# B&R Automation Studio project OpcUaSample410_BrbLibUa103 (part 14)

#### BrbUaRsGetEvent.c
```c
#include <bur/plctypes.h>
#ifdef __cplusplus
	extern "C"
	{
#endif

#include "BrbLibUa.h"
#include <string.h>
#include <AnsiCFunc.h>

#ifdef __cplusplus
	};
#endif

// NOLINTBEGIN(readability-*, bugprone-easily-swappable-parameters, bugprone-branch-clone, clang-diagnostic-invalid-utf8, clang-diagnostic-invalid-source-encoding, clang-diagnostic-pointer-arith, clang-diagnostic-strict-prototypes, hicpp-uppercase-literal-suffix, cppcoreguidelines-*, performance-*)

/* Gibt ein ermitteltes Event zurück */
unsigned short BrbUaRsGetEvent(struct BrbUaRunServer_TYP* pRunServer, unsigned short nEventIndex, struct BrbUaRsEvent_TYP* pEvent, struct BrbUaRsEventIntern_TYP* pEventIntern)
{
	UINT nStatus = eBRB_ERR_NULL_POINTER;
	if(pRunServer != 0 && pEvent != 0)
	{
		memset(pEvent, 0, sizeof(BrbUaRsEvent_TYP));
		nStatus = eBRB_ERR_UA_NO_ELEMENTS;
		if(pRunServer->Events.nEventCount > 0 && pRunServer->Events.pEvents != 0)
		{
			nStatus = eBRB_ERR_UA_INVALID_INDEX;
			if(nEventIndex < pRunServer->Events.nEventCount)
			{
				nStatus = eBRB_ERR_OK;
				BrbUaRsEventIntern_TYP* pEventInternOri = ((BrbUaRsEventIntern_TYP*)pRunServer->Events.pEvents) + nEventIndex;
				pEvent->nFieldCount = pEventInternOri->nFieldCount;
				memcpy(&pEvent->TypeNodeId, &pEventInternOri->TypeNodeId, sizeof(UANodeID));
				if(pEventIntern != 0)
				{
					memcpy(pEventIntern, pEventInternOri, sizeof(BrbUaRsEventIntern_TYP));
				}
			}
		}
	}
	return nStatus;
}

// NOLINTEND(readability-*, bugprone-easily-swappable-parameters, bugprone-branch-clone, clang-diagnostic-invalid-utf8, clang-diagnostic-invalid-source-encoding, clang-diagnostic-pointer-arith, clang-diagnostic-strict-prototypes, hicpp-uppercase-literal-suffix, cppcoreguidelines-*, performance-*)
```

#### BrbUaRsGetEventField.c
```c
#include <bur/plctypes.h>
#ifdef __cplusplus
	extern "C"
	{
#endif

#include "BrbLibUa.h"
#include <string.h>
#include <AnsiCFunc.h>

#ifdef __cplusplus
	};
#endif

// NOLINTBEGIN(readability-*, bugprone-easily-swappable-parameters, bugprone-branch-clone, clang-diagnostic-invalid-utf8, clang-diagnostic-invalid-source-encoding, clang-diagnostic-pointer-arith, clang-diagnostic-strict-prototypes, hicpp-uppercase-literal-suffix, cppcoreguidelines-*, performance-*)

/* Gibt ein ermitteltes Field zurück */
unsigned short BrbUaRsGetEventField(struct BrbUaRunServer_TYP* pRunServer, unsigned short nEventIndex, unsigned short nEventFieldIndex, struct UaSrv_FireEventFieldType* pEventField)
{
	UINT nStatus = eBRB_ERR_NULL_POINTER;
	if(pRunServer != 0 && pEventField != 0)
	{
		memset(pEventField, 0, sizeof(UaSrv_FireEventFieldType));
		nStatus = eBRB_ERR_UA_NO_ELEMENTS;
		if(pRunServer->Events.nEventCount > 0 && pRunServer->Events.pEvents != 0)
		{
			nStatus = eBRB_ERR_UA_INVALID_INDEX;
			if(nEventIndex < pRunServer->Events.nEventCount)
			{
				nStatus = eBRB_ERR_UA_NO_ELEMENTS;
				BrbUaRsEventIntern_TYP* pEventIntern = ((BrbUaRsEventIntern_TYP*)pRunServer->Events.pEvents) + nEventIndex;
				if(pEventIntern->nFieldCount > 0 && pEventIntern->pFields)
				{
					nStatus = eBRB_ERR_UA_INVALID_INDEX;
					if(nEventFieldIndex < pEventIntern->nFieldCount)
					{
						nStatus = eBRB_ERR_OK;
						UaSrv_FireEventFieldType* pEventFieldOri = ((UaSrv_FireEventFieldType*)pEventIntern->pFields) + nEventFieldIndex;
						memcpy(pEventField, pEventFieldOri, sizeof(UaSrv_FireEventFieldType));
					}
				}
			}
		}
	}
	return nStatus;
}

// NOLINTEND(readability-*, bugprone-easily-swappable-parameters, bugprone-branch-clone, clang-diagnostic-invalid-utf8, clang-diagnostic-invalid-source-encoding, clang-diagnostic-pointer-arith, clang-diagnostic-strict-prototypes, hicpp-uppercase-literal-suffix, cppcoreguidelines-*, performance-*)
```

#### BrbUaRsMonitor.c
```c
#include <bur/plctypes.h>
#ifdef __cplusplus
	extern "C"
	{
#endif

#include "BrbLibUa.h"
#include <string.h>
#include <AnsiCFunc.h>

#ifdef __cplusplus
	};
#endif

// NOLINTBEGIN(readability-*, bugprone-easily-swappable-parameters, bugprone-branch-clone, clang-diagnostic-invalid-utf8, clang-diagnostic-invalid-source-encoding, clang-diagnostic-pointer-arith, clang-diagnostic-strict-prototypes, hicpp-uppercase-literal-suffix, cppcoreguidelines-*, performance-*)

/* Zeigt die Inhalte des internen Speichers */
unsigned short BrbUaRsMonitor(struct BrbUaRunServer_TYP* pRunServer, struct BrbUaRsMonitor_TYP* pMonitor)
{
	UINT nStatus = eBRB_ERR_NULL_POINTER;
	if(pRunServer != 0 && pMonitor != 0)
	{
		nStatus = eBRB_ERR_NOT_ENABLED;
		if(pMonitor->bEnable == 1)
		{
			nStatus = eBRB_ERR_OK;
			brsmemset((UDINT)&pMonitor->Namespace.Namespace, 0, sizeof(pMonitor->Namespace.Namespace));
			BrbUaRsGetNamespace(pRunServer, pMonitor->Namespace.nDatObjNamespaceIndex, &pMonitor->Namespace.Namespace);

			brsmemset((UDINT)&pMonitor->Event.Event, 0, sizeof(pMonitor->Event.Event));
			brsmemset((UDINT)&pMonitor->Event.EventIntern, 0, sizeof(pMonitor->Event.EventIntern));
			pMonitor->Event.nMonitorStatus = BrbUaRsGetEvent(pRunServer, pMonitor->Event.nEventIndex, &pMonitor->Event.Event, &pMonitor->Event.EventIntern);

			brsmemset((UDINT)&pMonitor->EventField.Field, 0, sizeof(pMonitor->EventField.Field));
			pMonitor->EventField.nMonitorStatus = BrbUaRsGetEventField(pRunServer, pMonitor->EventField.nEventIndex, pMonitor->EventField.nEventFieldIndex, &pMonitor->EventField.Field);
		}
		else
		{
			brsmemset((UDINT)&pMonitor->Namespace.Namespace, 0, sizeof(pMonitor->Namespace.Namespace));
			pMonitor->Event.nMonitorStatus = eBRB_ERR_NOT_ENABLED;
			brsmemset((UDINT)&pMonitor->Event.Event, 0, sizeof(pMonitor->Event.Event));
			brsmemset((UDINT)&pMonitor->Event.EventIntern, 0, sizeof(pMonitor->Event.EventIntern));
			pMonitor->EventField.nMonitorStatus = eBRB_ERR_NOT_ENABLED;
			brsmemset((UDINT)&pMonitor->EventField.Field, 0, sizeof(pMonitor->EventField.Field));
		}
		pMonitor->nMonitorStatus = nStatus;
	}
	return nStatus;
}

// NOLINTEND(readability-*, bugprone-easily-swappable-parameters, bugprone-branch-clone, clang-diagnostic-invalid-utf8, clang-diagnostic-invalid-source-encoding, clang-diagnostic-pointer-arith, clang-diagnostic-strict-prototypes, hicpp-uppercase-literal-suffix, cppcoreguidelines-*, performance-*)
```

- Project.language (not shown)

### ReadMe.txt
```
Die AS-Solution 'UnitTest' ist eine Unterstützung für wiederholbare Aufruf-Tests.
Dabei sind Test-Routinen implementiert, welche ihrerseits Bibliotheks-Funktionen mit definierten Eingangs-Werten aufrufen,
die zurückgegebenen Ausgänge prüfen und so einen Bericht erstellen. Entspricht ein Ausgang nicht dem erwarteten Ergebnis,
wird dies im Bericht vermerkt.
Das Aufrufen aller Test-Routinen kann mit wenigen Mausklicks ausgeführt werden. So kann nach Änderung oder Erweiterung einer
Funktion sehr schnell deren Kompatibilität und Funktionstüchtigkeit geprüft werden, was zu einer Erhöhung der SW-Qualität führt.
Für das Beispiel zur Nutzung der geprüften Bibliothek sind die UnitTests nicht von Belang.
```

### Package Logical/UnitTests/UnitTestLibraries - Libraries for asserts

### Library Logical/UnitTests/UnitTestLibraries/BrbAsserts (ANSIC) - Brb custom asserts

#### BrbAsserts.h - Include this file in programs using any of the asserts provided by this library
```c
/********************************************************************
 * COPYRIGHT -- Bernecker + Rainer
 ********************************************************************
 * Library: BrbAsserts
 * File: BrbAsserts.h
 * Author: Rainer Niedermeier
 *******************************************************************/

#include <bur/plctypes.h>
#include "UnitTest.h"

/* When this file is included the defines, makros  of the following header files should be provided as well:  */
#include "EqualBool.h"
#include "EqualDint.h"
#include "EqualUdint.h"
#include "EqualDtStruct.h"
#include "WithinUdint.h"
#include "WithinDint.h"
#include "MemContent.h"
#include "StringEndContent.h"
```

#### EqualBool.h
```c
/********************************************************************
 * COPYRIGHT -- Bernecker + Rainer
 ********************************************************************
 * Library: BrbAsserts
 * File: EqualBool.c
 * Author: Rainer Niedermeier
 *******************************************************************/

#include <bur/plctypes.h>
#include "UnitTest.h"

#ifdef __cplusplus
extern "C"
{
#endif

// NOLINTBEGIN(readability-*, bugprone-easily-swappable-parameters, clang-diagnostic-invalid-utf8, clang-diagnostic-invalid-source-encoding, clang-diagnostic-pointer-arith, clang-diagnostic-strict-prototypes, hicpp-uppercase-literal-suffix, cppcoreguidelines-*, performance-*, readability-avoid-const-params-in-decls)

/* Dummies for smart edit autocompletion.
See below for the real macros used by the compiler  */
#ifdef _SMART_EDIT_DUMMY_
	/* Returns true if they are equal. */
	BOOL BRB_ASSERT_EQUAL_BOOL(const BOOL expected, const BOOL actual);
#endif

/* Prototyping of functions.
These declaration of functions are used by the compiler to check number and type of arguments. */
BOOL brb_assertEqualBool(const BOOL expected, const BOOL actual, unsigned long line, const char *file);

/* Macros used in the test implementation.
The macro passes the location information to the implemented assert. */
#define BRB_ASSERT_EQUAL_BOOL(expected, actual) brb_assertEqualBool(expected, actual, (unsigned long) __LINE__, __FILE__)

// NOLINTEND(readability-*, bugprone-easily-swappable-parameters, clang-diagnostic-invalid-utf8, clang-diagnostic-invalid-source-encoding, clang-diagnostic-pointer-arith, clang-diagnostic-strict-prototypes, hicpp-uppercase-literal-suffix, cppcoreguidelines-*, performance-*, readability-avoid-const-params-in-decls)

#ifdef __cplusplus
};
#endif
```

#### EqualBool.c
```c
/********************************************************************
 * COPYRIGHT -- Bernecker + Rainer
 ********************************************************************
 * Library: BrbAsserts
 * File: EqualBool.c
 * Author: Rainer Niedermeier
 *******************************************************************/

#include <bur/plctypes.h>
#include "BrbAsserts.h"
#include "AsBrStr.h"
#include "BrbLib.h"

#define TRUE 1
#define FALSE 0

// NOLINTBEGIN(readability-*, bugprone-easily-swappable-parameters, bugprone-branch-clone, clang-diagnostic-invalid-utf8, clang-diagnostic-invalid-source-encoding, clang-diagnostic-pointer-arith, clang-diagnostic-strict-prototypes, clang-diagnostic-bad-function-cast, clang-analyzer-security.insecureAPI.*, hicpp-uppercase-literal-suffix, cppcoreguidelines-*, performance-*)
BOOL brb_assertEqualBool(const BOOL expected, const BOOL actual,
	unsigned long line, const char *file)
{
	STRING buffer[100];
	STRING numbuf[15];
	BOOL result = TRUE;
	if(expected == actual)
	{
		addPassed("", line, file);
	}
	else
	{
		brsstrcpy((unsigned long) buffer, (unsigned long) "expected bool ");
		brsitoa((DINT)expected, (UDINT)&numbuf);
		brsstrcat((unsigned long) buffer, (unsigned long) numbuf);
		brsstrcat((unsigned long) buffer, (unsigned long) " was ");
		brsitoa((DINT)actual, (UDINT)&numbuf);
		brsstrcat((unsigned long) buffer, (unsigned long) numbuf);
		addFailure(buffer, line, file);
		result = FALSE;
	}
	return result;
}

// NOLINTEND(readability-*, bugprone-easily-swappable-parameters, bugprone-branch-clone, clang-diagnostic-invalid-utf8, clang-diagnostic-invalid-source-encoding, clang-diagnostic-pointer-arith, clang-diagnostic-strict-prototypes, clang-diagnostic-bad-function-cast, clang-analyzer-security.insecureAPI.*, hicpp-uppercase-literal-suffix, cppcoreguidelines-*, performance-*)
```

#### EqualDint.h
```c
/********************************************************************
 * COPYRIGHT -- Bernecker + Rainer
 ********************************************************************
 * Library: BrbAsserts
 * File: EqualDint.c
 * Author: Rainer Niedermeier
 *******************************************************************/

#include <bur/plctypes.h>
#include "UnitTest.h"

#ifdef __cplusplus
extern "C"
{
#endif

// NOLINTBEGIN(readability-*, bugprone-easily-swappable-parameters, clang-diagnostic-invalid-utf8, clang-diagnostic-invalid-source-encoding, clang-diagnostic-pointer-arith, clang-diagnostic-strict-prototypes, hicpp-uppercase-literal-suffix, cppcoreguidelines-*, performance-*, readability-avoid-const-params-in-decls)

/* Dummies for smart edit autocompletion.
See below for the real macros used by the compiler  */
#ifdef _SMART_EDIT_DUMMY_
	/* Returns true if they are equal. */
	BOOL BRB_ASSERT_EQUAL_DINT(const DINT expected, const DINT actual);
#endif

/* Prototyping of functions.
These declaration of functions are used by the compiler to check number and type of arguments. */
BOOL brb_assertEqualDint(const DINT expected, const DINT actual, unsigned long line, const char *file);

/* Macros used in the test implementation.
The macro passes the location information to the implemented assert. */
#define BRB_ASSERT_EQUAL_DINT(expected, actual) brb_assertEqualDint(expected, actual, (unsigned long) __LINE__, __FILE__)

// NOLINTEND(readability-*, bugprone-easily-swappable-parameters, clang-diagnostic-invalid-utf8, clang-diagnostic-invalid-source-encoding, clang-diagnostic-pointer-arith, clang-diagnostic-strict-prototypes, hicpp-uppercase-literal-suffix, cppcoreguidelines-*, performance-*, readability-avoid-const-params-in-decls)

#ifdef __cplusplus
};
#endif
```

#### EqualDint.c
```c
/********************************************************************
 * COPYRIGHT -- Bernecker + Rainer
 ********************************************************************
 * Library: BrbAsserts
 * File: EqualDint.c
 * Author: Rainer Niedermeier
 *******************************************************************/

#include <bur/plctypes.h>
#include "BrbAsserts.h"
#include "AsBrStr.h"
#include "BrbLib.h"

#define TRUE 1
#define FALSE 0

// NOLINTBEGIN(readability-*, bugprone-easily-swappable-parameters, bugprone-branch-clone, clang-diagnostic-invalid-utf8, clang-diagnostic-invalid-source-encoding, clang-diagnostic-pointer-arith, clang-diagnostic-strict-prototypes, clang-diagnostic-bad-function-cast, clang-analyzer-security.insecureAPI.*, hicpp-uppercase-literal-suffix, cppcoreguidelines-*, performance-*)
BOOL brb_assertEqualDint(const DINT expected, const DINT actual,
	unsigned long line, const char *file)
{
	STRING buffer[100];
	STRING numbuf[15];
	BOOL result = TRUE;
	if(expected == actual)
	{
		addPassed("", line, file);
	}
	else
	{
		brsstrcpy((unsigned long) buffer, (unsigned long) "expected dint ");
		brsitoa((DINT)expected, (UDINT)&numbuf);
		brsstrcat((unsigned long) buffer, (unsigned long) numbuf);
		brsstrcat((unsigned long) buffer, (unsigned long) " was ");
		brsitoa((DINT)actual, (UDINT)&numbuf);
		brsstrcat((unsigned long) buffer, (unsigned long) numbuf);
		addFailure(buffer, line, file);
		result = FALSE;
	}
	return result;
}

// NOLINTEND(readability-*, bugprone-easily-swappable-parameters, bugprone-branch-clone, clang-diagnostic-invalid-utf8, clang-diagnostic-invalid-source-encoding, clang-diagnostic-pointer-arith, clang-diagnostic-strict-prototypes, clang-diagnostic-bad-function-cast, clang-analyzer-security.insecureAPI.*, hicpp-uppercase-literal-suffix, cppcoreguidelines-*, performance-*)
```

#### EqualUdint.h
```c
/********************************************************************
 * COPYRIGHT -- Bernecker + Rainer
 ********************************************************************
 * Library: BrbAsserts
 * File: EqualUdint.c
 * Author: Rainer Niedermeier
 *******************************************************************/

#include <bur/plctypes.h>
#include "UnitTest.h"

#ifdef __cplusplus
extern "C"
{
#endif

// NOLINTBEGIN(readability-*, bugprone-easily-swappable-parameters, clang-diagnostic-invalid-utf8, clang-diagnostic-invalid-source-encoding, clang-diagnostic-pointer-arith, clang-diagnostic-strict-prototypes, hicpp-uppercase-literal-suffix, cppcoreguidelines-*, performance-*, readability-avoid-const-params-in-decls)

/* Dummies for smart edit autocompletion.
See below for the real macros used by the compiler  */
#ifdef _SMART_EDIT_DUMMY_
	/* Returns true if they are equal. */
	BOOL BRB_ASSERT_EQUAL_UDINT(const UDINT expected, const UDINT actual);
#endif

/* Prototyping of functions.
These declaration of functions are used by the compiler to check number and type of arguments. */
BOOL brb_assertEqualUdint(const UDINT expected, const UDINT actual, unsigned long line, const char *file);

/* Macros used in the test implementation.
The macro passes the location information to the implemented assert. */
#define BRB_ASSERT_EQUAL_UDINT(expected, actual) brb_assertEqualUdint(expected, actual, (unsigned long) __LINE__, __FILE__)

// NOLINTEND(readability-*, bugprone-easily-swappable-parameters, clang-diagnostic-invalid-utf8, clang-diagnostic-invalid-source-encoding, clang-diagnostic-pointer-arith, clang-diagnostic-strict-prototypes, hicpp-uppercase-literal-suffix, cppcoreguidelines-*, performance-*, readability-avoid-const-params-in-decls)

#ifdef __cplusplus
};
#endif
```

#### EqualUdint.c
```c
/********************************************************************
 * COPYRIGHT -- Bernecker + Rainer
 ********************************************************************
 * Library: BrbAsserts
 * File: EqualUdint.c
 * Author: Rainer Niedermeier
 *******************************************************************/

#include <bur/plctypes.h>
#include "BrbAsserts.h"
#include "AsBrStr.h"
#include "BrbLib.h"

#define TRUE 1
#define FALSE 0

// NOLINTBEGIN(readability-*, bugprone-easily-swappable-parameters, bugprone-branch-clone, clang-diagnostic-invalid-utf8, clang-diagnostic-invalid-source-encoding, clang-diagnostic-pointer-arith, clang-diagnostic-strict-prototypes, clang-diagnostic-bad-function-cast, clang-analyzer-security.insecureAPI.*, hicpp-uppercase-literal-suffix, cppcoreguidelines-*, performance-*)
BOOL brb_assertEqualUdint(const UDINT expected, const UDINT actual,
	unsigned long line, const char *file)
{
	STRING buffer[100];
	STRING numbuf[15];

	BOOL result = TRUE;
	if(expected == actual)
	{
		addPassed("", line, file);
	}
	else
	{
		brsstrcpy((unsigned long) buffer, (unsigned long) "expected udint ");
		BrbUdintToAscii(expected, numbuf);
		brsstrcat((unsigned long) buffer, (unsigned long) numbuf);
		brsstrcat((unsigned long) buffer, (unsigned long) " was ");
		BrbUdintToAscii(actual, numbuf);
		brsstrcat((unsigned long) buffer, (unsigned long) numbuf);
		addFailure(buffer, line, file);
		result = FALSE;
	}
	return result;
}

// NOLINTEND(readability-*, bugprone-easily-swappable-parameters, bugprone-branch-clone, clang-diagnostic-invalid-utf8, clang-diagnostic-invalid-source-encoding, clang-diagnostic-pointer-arith, clang-diagnostic-strict-prototypes, clang-diagnostic-bad-function-cast, clang-analyzer-security.insecureAPI.*, hicpp-uppercase-literal-suffix, cppcoreguidelines-*, performance-*)
```

#### EqualDtStruct.h
```c
/********************************************************************
 * COPYRIGHT -- Bernecker + Rainer
 ********************************************************************
 * Library: BrbAsserts
 * File: Equal_Udint.h
 * Author: Rainer Niedermeier
 *******************************************************************/

#include <bur/plctypes.h>
#include "UnitTest.h"
#include "AsTime.h" // NOLINT(clang-diagnostic-nonportable-system-include-path)

#ifdef __cplusplus
extern "C"
{
#endif

// NOLINTBEGIN(readability-*, bugprone-easily-swappable-parameters, clang-diagnostic-invalid-utf8, clang-diagnostic-invalid-source-encoding, clang-diagnostic-pointer-arith, clang-diagnostic-strict-prototypes, hicpp-uppercase-literal-suffix, cppcoreguidelines-*, performance-*, readability-avoid-const-params-in-decls)

/* Dummies for smart edit autocompletion.
See below for the real macros used by the compiler  */
#ifdef _SMART_EDIT_DUMMY_
	/* Returns true if they are equal. */
	BOOL BRB_ASSERT_EQUAL_DTSTRUCT(const UINT expectedYear, const USINT expectedMonth, const USINT expectedDay, const USINT expectedWeekday, const USINT expectedHour, const USINT expectedMinute, const USINT expectedSecond, const USINT expectedMilliSecond, const USINT expectedMicroSecond, const DTStructure* actual);
#endif

/* Prototyping of functions.
These declaration of functions are used by the compiler to check number and type of arguments. */
BOOL brb_assertEqualDtStruct(const UINT expectedYear, const USINT expectedMonth, const USINT expectedDay, const USINT expectedWeekday, const USINT expectedHour, const USINT expectedMinute, const USINT expectedSecond, const UINT expectedMilliSecond, const UINT expectedMicroSecond, const DTStructure* actual, unsigned long line, const char *file);

/* Macros used in the test implementation.
The macro passes the location information to the implemented assert. */
#define BRB_ASSERT_EQUAL_DTSTRUCT(expectedYear, expectedMonth, expectedDay, expectedWeekday, expectedHour, expectedMinute, expectedSecond, expectedMilliSecond, expectedMicroSecond, actual) brb_assertEqualDtStruct(expectedYear, expectedMonth, expectedDay, expectedWeekday, expectedHour, expectedMinute, expectedSecond, expectedMilliSecond, expectedMicroSecond, actual, (unsigned long) __LINE__, __FILE__)

// NOLINTEND(readability-*, bugprone-easily-swappable-parameters, clang-diagnostic-invalid-utf8, clang-diagnostic-invalid-source-encoding, clang-diagnostic-pointer-arith, clang-diagnostic-strict-prototypes, hicpp-uppercase-literal-suffix, cppcoreguidelines-*, performance-*, readability-avoid-const-params-in-decls)

#ifdef __cplusplus
};
#endif
```

#### EqualDtStruct.c
```c
/********************************************************************
 * COPYRIGHT -- Bernecker + Rainer
 ********************************************************************
 * Library: BrbAsserts
 * File: Equal_Udint.c
 * Author: Rainer Niedermeier
 *******************************************************************/

#include <bur/plctypes.h>
#include "AsBrStr.h"
#include "EqualDtStruct.h"

#define TRUE 1
#define FALSE 0

// NOLINTBEGIN(readability-*, bugprone-easily-swappable-parameters, bugprone-branch-clone, clang-diagnostic-invalid-utf8, clang-diagnostic-invalid-source-encoding, clang-diagnostic-pointer-arith, clang-diagnostic-strict-prototypes, clang-diagnostic-bad-function-cast, clang-analyzer-security.insecureAPI.*, hicpp-uppercase-literal-suffix, cppcoreguidelines-*, performance-*)
BOOL brb_assertEqualDtStruct(const UINT expectedYear, const USINT expectedMonth, const USINT expectedDay, const USINT expectedWeekday,
														const USINT expectedHour, const USINT expectedMinute, const USINT expectedSecond,
														const UINT expectedMilliSecond, const UINT expectedMicroSecond,
														const DTStructure* actual,
                         		unsigned long line, const char *file)
{
	STRING buffer[100];
	STRING numbuf[15];
	BOOL result = TRUE;
	// year
	if(expectedYear == actual->year)
	{
		addPassed("", line, file);
	}
	else
	{
		brsstrcpy((unsigned long) buffer, (unsigned long) "expected year ");
		brsitoa((int)expectedYear, (unsigned long)numbuf);
		brsstrcat((unsigned long) buffer, (unsigned long) numbuf);
		brsstrcat((unsigned long) buffer, (unsigned long) " was ");
		brsitoa((int)actual->year, (unsigned long)numbuf);
		brsstrcat((unsigned long) buffer, (unsigned long) numbuf);
		addFailure(buffer, line, file);
		result = FALSE;
	}
	// month
	if(expectedMonth == actual->month)
	{
		addPassed("", line, file);
	}
	else
	{
		brsstrcpy((unsigned long) buffer, (unsigned long) "expected month ");
		brsitoa((int)expectedMonth, (unsigned long)numbuf);
		brsstrcat((unsigned long) buffer, (unsigned long) numbuf);
		brsstrcat((unsigned long) buffer, (unsigned long) " was ");
		brsitoa((int)actual->month, (unsigned long)numbuf);
		brsstrcat((unsigned long) buffer, (unsigned long) numbuf);
		addFailure(buffer, line, file);
		result = FALSE;
	}
	// day
	if(expectedDay == actual->day)
	{
		addPassed("", line, file);
	}
	else
	{
		brsstrcpy((unsigned long) buffer, (unsigned long) "expected day ");
		brsitoa((int)expectedDay, (unsigned long)numbuf);
		brsstrcat((unsigned long) buffer, (unsigned long) numbuf);
		brsstrcat((unsigned long) buffer, (unsigned long) " was ");
		brsitoa((int)actual->day, (unsigned long)numbuf);
		brsstrcat((unsigned long) buffer, (unsigned long) numbuf);
		addFailure(buffer, line, file);
		result = FALSE;
	}
	// weekday
	if(expectedWeekday == actual->wday)
	{
		addPassed("", line, file);
	}
	else
	{
		brsstrcpy((unsigned long) buffer, (unsigned long) "expected weekday ");
		brsitoa((int)expectedWeekday, (unsigned long)numbuf);
		brsstrcat((unsigned long) buffer, (unsigned long) numbuf);
		brsstrcat((unsigned long) buffer, (unsigned long) " was ");
		brsitoa((int)actual->wday, (unsigned long)numbuf);
		brsstrcat((unsigned long) buffer, (unsigned long) numbuf);
		addFailure(buffer, line, file);
		result = FALSE;
	}
	// hour
	if(expectedHour == actual->hour)
	{
		addPassed("", line, file);
	}
	else
	{
		brsstrcpy((unsigned long) buffer, (unsigned long) "expected hour ");
		brsitoa((int)expectedHour, (unsigned long)numbuf);
		brsstrcat((unsigned long) buffer, (unsigned long) numbuf);
		brsstrcat((unsigned long) buffer, (unsigned long) " was ");
		brsitoa((int)actual->hour, (unsigned long)numbuf);
		brsstrcat((unsigned long) buffer, (unsigned long) numbuf);
		addFailure(buffer, line, file);
		result = FALSE;
	}
	// minute
	if(expectedMinute == actual->minute)
	{
		addPassed("", line, file);
	}
	else
	{
		brsstrcpy((unsigned long) buffer, (unsigned long) "expected minute ");
		brsitoa((int)expectedMinute, (unsigned long)numbuf);
		brsstrcat((unsigned long) buffer, (unsigned long) numbuf);
		brsstrcat((unsigned long) buffer, (unsigned long) " was ");
		brsitoa((int)actual->minute, (unsigned long)numbuf);
		brsstrcat((unsigned long) buffer, (unsigned long) numbuf);
		addFailure(buffer, line, file);
		result = FALSE;
	}
	// second
	if(expectedSecond == actual->second)
	{
		addPassed("", line, file);
	}
	else
	{
		brsstrcpy((unsigned long) buffer, (unsigned long) "expected second ");
		brsitoa((int)expectedSecond, (unsigned long)numbuf);
		brsstrcat((unsigned long) buffer, (unsigned long) numbuf);
		brsstrcat((unsigned long) buffer, (unsigned long) " was ");
		brsitoa((int)actual->second, (unsigned long)numbuf);
		brsstrcat((unsigned long) buffer, (unsigned long) numbuf);
		addFailure(buffer, line, file);
		result = FALSE;
	}
	// millisecond
	if(expectedMilliSecond == actual->millisec)
	{
		addPassed("", line, file);
	}
	else
	{
		brsstrcpy((unsigned long) buffer, (unsigned long) "expected millisecond ");
		brsitoa((int)expectedMilliSecond, (unsigned long)numbuf);
		brsstrcat((unsigned long) buffer, (unsigned long) numbuf);
		brsstrcat((unsigned long) buffer, (unsigned long) " was ");
		brsitoa((int)actual->millisec, (unsigned long)numbuf);
		brsstrcat((unsigned long) buffer, (unsigned long) numbuf);
		addFailure(buffer, line, file);
		result = FALSE;
	}
	// microsecond
	if(expectedMicroSecond == actual->microsec)
	{
		addPassed("", line, file);
	}
	else
	{
		brsstrcpy((unsigned long) buffer, (unsigned long) "expected microsecond ");
		brsitoa((int)expectedMicroSecond, (unsigned long)numbuf);
		brsstrcat((unsigned long) buffer, (unsigned long) numbuf);
		brsstrcat((unsigned long) buffer, (unsigned long) " was ");
		brsitoa((int)actual->microsec, (unsigned long)numbuf);
		brsstrcat((unsigned long) buffer, (unsigned long) numbuf);
		addFailure(buffer, line, file);
		result = FALSE;
	}
	return result;
}

// NOLINTEND(readability-*, bugprone-easily-swappable-parameters, bugprone-branch-clone, clang-diagnostic-invalid-utf8, clang-diagnostic-invalid-source-encoding, clang-diagnostic-pointer-arith, clang-diagnostic-strict-prototypes, clang-diagnostic-bad-function-cast, clang-analyzer-security.insecureAPI.*, hicpp-uppercase-literal-suffix, cppcoreguidelines-*, performance-*)
```

#### WithinUdint.h
```c
/********************************************************************
 * COPYRIGHT -- Bernecker + Rainer
 ********************************************************************
 * Library: BrbAsserts
 * File: Equal_Udint.h
 * Author: Rainer Niedermeier
 *******************************************************************/

#include <bur/plctypes.h>
#include "UnitTest.h"

#ifdef __cplusplus
extern "C"
{
#endif

// NOLINTBEGIN(readability-*, bugprone-easily-swappable-parameters, clang-diagnostic-invalid-utf8, clang-diagnostic-invalid-source-encoding, clang-diagnostic-pointer-arith, clang-diagnostic-strict-prototypes, hicpp-uppercase-literal-suffix, cppcoreguidelines-*, performance-*, readability-avoid-const-params-in-decls)

/* Dummies for smart edit autocompletion.
See below for the real macros used by the compiler  */
#ifdef _SMART_EDIT_DUMMY_
	/* Returns true if they are equal. */
	BOOL BRB_ASSERT_WITHIN_UDINT(const UDINT min, const UDINT max, const UDINT actual);
#endif

/* Prototyping of functions.
These declaration of functions are used by the compiler to check number and type of arguments. */
BOOL brb_assertWithinUdint(const UDINT min, const UDINT max, const UDINT actual, unsigned long line, const char *file);

/* Macros used in the test implementation.
The macro passes the location information to the implemented assert. */
#define BRB_ASSERT_WITHIN_UDINT(min, max, actual) brb_assertWithinUdint(min, max, actual, (unsigned long) __LINE__, __FILE__)

// NOLINTEND(readability-*, bugprone-easily-swappable-parameters, clang-diagnostic-invalid-utf8, clang-diagnostic-invalid-source-encoding, clang-diagnostic-pointer-arith, clang-diagnostic-strict-prototypes, hicpp-uppercase-literal-suffix, cppcoreguidelines-*, performance-*, readability-avoid-const-params-in-decls)

#ifdef __cplusplus
};
#endif
```

#### WithinUdint.c
```c
/********************************************************************
 * COPYRIGHT -- Bernecker + Rainer
 ********************************************************************
 * Library: BrbAsserts
 * File: Equal_Udint.c
 * Author: Rainer Niedermeier
 *******************************************************************/

#include <bur/plctypes.h>
#include "AsBrStr.h"
#include "BrbLib.h"
#include "WithinUdint.h"

#define TRUE 1
#define FALSE 0

// NOLINTBEGIN(readability-*, bugprone-easily-swappable-parameters, bugprone-branch-clone, clang-diagnostic-invalid-utf8, clang-diagnostic-invalid-source-encoding, clang-diagnostic-pointer-arith, clang-diagnostic-strict-prototypes, clang-diagnostic-bad-function-cast, clang-analyzer-security.insecureAPI.*, hicpp-uppercase-literal-suffix, cppcoreguidelines-*, performance-*)
BOOL brb_assertWithinUdint(const UDINT min, const UDINT max, const UDINT actual,
                         		unsigned long line, const char *file)
{
	STRING buffer[100];
	STRING numbuf[15];
	BOOL result = TRUE;
	if(actual >= min && actual <= max)
	{
		addPassed("", line, file);
	}
	else
	{
		brsstrcpy((unsigned long) buffer, (unsigned long) "expected udint ");
		BrbUdintToAscii(actual, numbuf);
		brsstrcat((unsigned long) buffer, (unsigned long) numbuf);
		brsstrcat((unsigned long) buffer, (unsigned long) " was outside range (min=");
		BrbUdintToAscii(min, numbuf);
		brsstrcat((unsigned long) buffer, (unsigned long) numbuf);
		brsstrcat((unsigned long) buffer, (unsigned long) ", max=");
		BrbUdintToAscii(max, numbuf);
		brsstrcat((unsigned long) buffer, (unsigned long) numbuf);
		brsstrcat((unsigned long) buffer, (unsigned long) ")");
		addFailure(buffer, line, file);
		result = FALSE;
	}
	return result;
}

// NOLINTEND(readability-*, bugprone-easily-swappable-parameters, bugprone-branch-clone, clang-diagnostic-invalid-utf8, clang-diagnostic-invalid-source-encoding, clang-diagnostic-pointer-arith, clang-diagnostic-strict-prototypes, clang-diagnostic-bad-function-cast, clang-analyzer-security.insecureAPI.*, hicpp-uppercase-literal-suffix, cppcoreguidelines-*, performance-*)
```

#### WithinDint.h
```c
/********************************************************************
 * COPYRIGHT -- Bernecker + Rainer
 ********************************************************************
 * Library: BrbAsserts
 * File: Equal_Dint.h
 * Author: Rainer Niedermeier
 *******************************************************************/

#include <bur/plctypes.h>
#include "UnitTest.h"

#ifdef __cplusplus
extern "C"
{
#endif

// NOLINTBEGIN(readability-*, bugprone-easily-swappable-parameters, clang-diagnostic-invalid-utf8, clang-diagnostic-invalid-source-encoding, clang-diagnostic-pointer-arith, clang-diagnostic-strict-prototypes, hicpp-uppercase-literal-suffix, cppcoreguidelines-*, performance-*, readability-avoid-const-params-in-decls)

/* Dummies for smart edit autocompletion.
See below for the real macros used by the compiler  */
#ifdef _SMART_EDIT_DUMMY_
	/* Returns true if they are equal. */
	BOOL BRB_ASSERT_WITHIN_DINT(const DINT min, const DINT max, const DINT actual);
#endif

/* Prototyping of functions.
These declaration of functions are used by the compiler to check number and type of arguments. */
BOOL brb_assertWithinDint(const DINT min, const DINT max, const DINT actual, unsigned long line, const char *file);

/* Macros used in the test implementation.
The macro passes the location information to the implemented assert. */
#define BRB_ASSERT_WITHIN_DINT(min, max, actual) brb_assertWithinDint(min, max, actual, (unsigned long) __LINE__, __FILE__)

// NOLINTEND(readability-*, bugprone-easily-swappable-parameters, clang-diagnostic-invalid-utf8, clang-diagnostic-invalid-source-encoding, clang-diagnostic-pointer-arith, clang-diagnostic-strict-prototypes, hicpp-uppercase-literal-suffix, cppcoreguidelines-*, performance-*, readability-avoid-const-params-in-decls)

#ifdef __cplusplus
};
#endif
```

#### WithinDint.c
```c
/********************************************************************
 * COPYRIGHT -- Bernecker + Rainer
 ********************************************************************
 * Library: BrbAsserts
 * File: Equal_Dint.c
 * Author: Rainer Niedermeier
 *******************************************************************/

#include <bur/plctypes.h>
#include "AsBrStr.h"
#include "BrbLib.h"
#include "WithinDint.h"

#define TRUE 1
#define FALSE 0

// NOLINTBEGIN(readability-*, bugprone-easily-swappable-parameters, bugprone-branch-clone, clang-diagnostic-invalid-utf8, clang-diagnostic-invalid-source-encoding, clang-diagnostic-pointer-arith, clang-diagnostic-strict-prototypes, clang-diagnostic-bad-function-cast, clang-analyzer-security.insecureAPI.*, hicpp-uppercase-literal-suffix, cppcoreguidelines-*, performance-*)
BOOL brb_assertWithinDint(const DINT min, const DINT max, const DINT actual,
                         		unsigned long line, const char *file)
{
	STRING buffer[100];
	STRING numbuf[15];
	BOOL result = TRUE;
	if(actual >= min && actual <= max)
	{
		addPassed("", line, file);
	}
	else
	{
		brsstrcpy((unsigned long) buffer, (unsigned long) "expected dint ");
		brsitoa((int)actual, (unsigned long)numbuf);
		brsstrcat((unsigned long) buffer, (unsigned long) numbuf);
		brsstrcat((unsigned long) buffer, (unsigned long) " was outside range (min=");
		brsitoa((int)min, (unsigned long)numbuf);
		brsstrcat((unsigned long) buffer, (unsigned long) numbuf);
		brsstrcat((unsigned long) buffer, (unsigned long) ", max=");
		brsitoa((int)max, (unsigned long)numbuf);
		brsstrcat((unsigned long) buffer, (unsigned long) numbuf);
		brsstrcat((unsigned long) buffer, (unsigned long) ")");
		addFailure(buffer, line, file);
		result = FALSE;
	}
	return result;
}

// NOLINTEND(readability-*, bugprone-easily-swappable-parameters, bugprone-branch-clone, clang-diagnostic-invalid-utf8, clang-diagnostic-invalid-source-encoding, clang-diagnostic-pointer-arith, clang-diagnostic-strict-prototypes, clang-diagnostic-bad-function-cast, clang-analyzer-security.insecureAPI.*, hicpp-uppercase-literal-suffix, cppcoreguidelines-*, performance-*)
```

#### MemContent.h
```c
/********************************************************************
 * COPYRIGHT -- Bernecker + Rainer
 ********************************************************************
 * Library: BrbAsserts
 * File: MemContent.h
 * Author: Rainer Niedermeier
 *******************************************************************/

#include <bur/plctypes.h>
#include "UnitTest.h"

#ifdef __cplusplus
extern "C"
{
#endif

// NOLINTBEGIN(readability-*, bugprone-easily-swappable-parameters, clang-diagnostic-invalid-utf8, clang-diagnostic-invalid-source-encoding, clang-diagnostic-pointer-arith, clang-diagnostic-strict-prototypes, hicpp-uppercase-literal-suffix, cppcoreguidelines-*, performance-*, readability-avoid-const-params-in-decls)

/* Dummies for smart edit autocompletion.
See below for the real macros used by the compiler  */
#ifdef _SMART_EDIT_DUMMY_
	/* Returns true if they are equal. */
	BOOL BRB_ASSERT_MEM_CONTENT(const UDINT mem, const USINT content, const UDINT size);
#endif

/* Prototyping of functions.
These declaration of functions are used by the compiler to check number and type of arguments. */
BOOL brb_assertMemContent(const UDINT mem, const USINT content, const UDINT size, unsigned long line, const char *file);

/* Macros used in the test implementation.
The macro passes the location information to the implemented assert. */
#define BRB_ASSERT_MEM_CONTENT(mem, content, size) brb_assertMemContent(mem, content, size, (unsigned long) __LINE__, __FILE__)

// NOLINTEND(readability-*, bugprone-easily-swappable-parameters, clang-diagnostic-invalid-utf8, clang-diagnostic-invalid-source-encoding, clang-diagnostic-pointer-arith, clang-diagnostic-strict-prototypes, hicpp-uppercase-literal-suffix, cppcoreguidelines-*, performance-*, readability-avoid-const-params-in-decls)

#ifdef __cplusplus
};
#endif
```

#### MemContent.c
```c
/********************************************************************
 * COPYRIGHT -- Bernecker + Rainer
 ********************************************************************
 * Library: BrbAsserts
 * File: MemContent.c
 * Author: Rainer Niedermeier
 *******************************************************************/

#include <bur/plctypes.h>
#include "AsBrStr.h"
#include "BrbLib.h"
#include "WithinDint.h"

#define TRUE 1
#define FALSE 0

// NOLINTBEGIN(readability-*, bugprone-easily-swappable-parameters, bugprone-branch-clone, clang-diagnostic-invalid-utf8, clang-diagnostic-invalid-source-encoding, clang-diagnostic-pointer-arith, clang-diagnostic-strict-prototypes, clang-diagnostic-bad-function-cast, clang-analyzer-security.insecureAPI.*, hicpp-uppercase-literal-suffix, cppcoreguidelines-*, performance-*)
BOOL brb_assertMemContent(const UDINT mem, const USINT content, const UDINT size,
                         		unsigned long line, const char *file)
{
	STRING buffer[100];
	STRING numbuf[15];
	BOOL result = TRUE;
	UDINT index = 0;
	for(index=0; index<size; index++)
	{
		USINT* pointer = ((USINT*)mem) + index;
		USINT value = *pointer;
		if(value != content)
		{
			brsstrcpy((unsigned long) buffer, (unsigned long) "expected mem content [");
			brsitoa((int)index, (unsigned long)numbuf);
			brsstrcat((unsigned long) buffer, (unsigned long) numbuf);
			brsstrcat((unsigned long) buffer, (unsigned long) "] is ");
			brsitoa((int)value, (unsigned long)numbuf);
			brsstrcat((unsigned long) buffer, (unsigned long) numbuf);
			brsstrcat((unsigned long) buffer, (unsigned long) ", not ");
			brsitoa((int)content, (unsigned long)numbuf);
			brsstrcat((unsigned long) buffer, (unsigned long) numbuf);
			addFailure(buffer, line, file);
			result = FALSE;
		}
	}
	if(result == TRUE)
	{
		addPassed("", line, file);
	}
	return result;
}

// NOLINTEND(readability-*, bugprone-easily-swappable-parameters, bugprone-branch-clone, clang-diagnostic-invalid-utf8, clang-diagnostic-invalid-source-encoding, clang-diagnostic-pointer-arith, clang-diagnostic-strict-prototypes, clang-diagnostic-bad-function-cast, clang-analyzer-security.insecureAPI.*, hicpp-uppercase-literal-suffix, cppcoreguidelines-*, performance-*)
```

#### StringEndContent.h
```c
/********************************************************************
 * COPYRIGHT -- Bernecker + Rainer
 ********************************************************************
 * Library: BrbAsserts
 * File: StringEndContent.h
 * Author: Rainer Niedermeier
 *******************************************************************/

#include <bur/plctypes.h>
#include "UnitTest.h"

#ifdef __cplusplus
extern "C"
{
#endif

// NOLINTBEGIN(readability-*, bugprone-easily-swappable-parameters, clang-diagnostic-invalid-utf8, clang-diagnostic-invalid-source-encoding, clang-diagnostic-pointer-arith, clang-diagnostic-strict-prototypes, hicpp-uppercase-literal-suffix, cppcoreguidelines-*, performance-*, readability-avoid-const-params-in-decls)

/* Dummies for smart edit autocompletion.
See below for the real macros used by the compiler  */
#ifdef _SMART_EDIT_DUMMY_
	/* Returns true if they are equal. */
	BOOL BRB_ASSERT_STRING_END_CONTENT(const UDINT mem, const USINT content, const UDINT size, const UDINT start);
#endif

/* Prototyping of functions.
These declaration of functions are used by the compiler to check number and type of arguments. */
BOOL brb_assertStringEndContent(const UDINT mem, const USINT content, const UDINT size, const UDINT start, unsigned long line, const char *file);

/* Macros used in the test implementation.
The macro passes the location information to the implemented assert. */
#define BRB_ASSERT_STRING_END_CONTENT(mem, content, size, start) brb_assertStringEndContent(mem, content, size, start, (unsigned long) __LINE__, __FILE__)

// NOLINTEND(readability-*, bugprone-easily-swappable-parameters, clang-diagnostic-invalid-utf8, clang-diagnostic-invalid-source-encoding, clang-diagnostic-pointer-arith, clang-diagnostic-strict-prototypes, hicpp-uppercase-literal-suffix, cppcoreguidelines-*, performance-*, readability-avoid-const-params-in-decls)

#ifdef __cplusplus
};
#endif
```

#### StringEndContent.c
```c
/********************************************************************
 * COPYRIGHT -- Bernecker + Rainer
 ********************************************************************
 * Library: BrbAsserts
 * File: StringEndContent.c
 * Author: Rainer Niedermeier
 *******************************************************************/

#include <bur/plctypes.h>
#include "AsBrStr.h"
#include "BrbLib.h"
#include "WithinDint.h"

#define TRUE 1
#define FALSE 0

// NOLINTBEGIN(readability-*, bugprone-easily-swappable-parameters, bugprone-branch-clone, clang-diagnostic-invalid-utf8, clang-diagnostic-invalid-source-encoding, clang-diagnostic-pointer-arith, clang-diagnostic-strict-prototypes, clang-diagnostic-bad-function-cast, clang-analyzer-security.insecureAPI.*, hicpp-uppercase-literal-suffix, cppcoreguidelines-*, performance-*)
BOOL brb_assertStringEndContent(const UDINT mem, const USINT content, const UDINT size, const UDINT start,
                         		unsigned long line, const char *file)
{
	STRING buffer[100];
	STRING numbuf[15];
	BOOL result = TRUE;
	UDINT index = 0;
	for(index=0; index<size; index++)
	{
		if(index>=start)
		{
			USINT* pointer = ((USINT*)mem) + index;
			USINT value = *pointer;
			if(value != content)
			{
				brsstrcpy((unsigned long) buffer, (unsigned long) "expected string end content [");
				brsitoa((int)index, (unsigned long)numbuf);
				brsstrcat((unsigned long) buffer, (unsigned long) numbuf);
				brsstrcat((unsigned long) buffer, (unsigned long) "] is ");
				brsitoa((int)value, (unsigned long)numbuf);
				brsstrcat((unsigned long) buffer, (unsigned long) numbuf);
				brsstrcat((unsigned long) buffer, (unsigned long) ", not ");
				brsitoa((int)content, (unsigned long)numbuf);
				brsstrcat((unsigned long) buffer, (unsigned long) numbuf);
				addFailure(buffer, line, file);
				result = FALSE;
			}
		}
	}
	if(result == TRUE)
	{
		addPassed("", line, file);
	}
	return result;
}

// NOLINTEND(readability-*, bugprone-easily-swappable-parameters, bugprone-branch-clone, clang-diagnostic-invalid-utf8, clang-diagnostic-invalid-source-encoding, clang-diagnostic-pointer-arith, clang-diagnostic-strict-prototypes, clang-diagnostic-bad-function-cast, clang-analyzer-security.insecureAPI.*, hicpp-uppercase-literal-suffix, cppcoreguidelines-*, performance-*)
```

### Program Logical/UnitTests/UtBrbUaTemplate (ANSIC) - UnitTests

#### variables.var - Name the suite and add PVs for the program
```iecst
(********************************************************************
 * COPYRIGHT --
 ********************************************************************
 * Program: utTemplate_automated
 * File: variables.var
 * Author: -
 * Created: -
 ********************************************************************
 * Local variables of program utTemplate_automated
 ********************************************************************)
(*Describe the test*)
VAR
	Testsuite : UtMgrTestSuite := (Name:='BrbUaTemplate',Description:='(Optional field)Template for use with helper tool. Reference or add this program in the package "TS_UnitTest_UpdateTestPrograms"',Type:=utMgrTEST_TYPE_C,MetaInformation:='(Optional field):To be filled');
END_VAR
(*Input variables for testing*)
(*Functionblock instances for testing*)
(*Output variables for testing*)
VAR
	uintOut0 : UINT := 0;
END_VAR
```

#### autoGeneratedFile.c - Auto generated code - list of all test sets in the program
```c
/*
B+R UnitTest: This is generated code.
Do not edit! Do not move!
Description: UnitTest Testprogramm infrastructure (List of TestSets).
LastUpdated: 2021-05-03 06:15:16Z
By B+R UnitTest Helper Version: 2.0.1.59
*/
#include "UnitTest.h"

UNITTEST_TESTSET_DECLARATION  Set_BrbTemplateFunc;

UNITTEST_TESTSET_FIXTURES(utTestSets)
{
	new_TestSet(Set_BrbTemplateFunc),
};
UNTITTEST_TESTSET_HANDLER();
```

#### Set_BrbUaTemplateFunc.c - Test set
```c
#include <bur/plctypes.h>

#ifdef _DEFAULT_INCLUDES
#include <AsDefault.h>
#endif

#include "UnitTest.h"
#include "BrbAsserts.h"
#include <string.h>

_TEST BrbXXX(void)
{
	// Init
	//memset(&xxx, 0, sizeof(xxx));
	//strcpy(stringIn0, "");

	// Call
	uintOut0 = 0;//BrbXXX();

	// Assert
	//TEST_ASSERT_EQUAL_INT(eBRB_ERR_NULL_POINTER, uintOut0);
	//TEST_ASSERT_EQUAL_STRING("", stringIn0);

	// Finished
	TEST_DONE;
}

/*
B+R UnitTest: This is generated code.
Do not edit! Do not move!
Description: UnitTest Testprogramm infrastructure (TestSet).
LastUpdated: 2021-05-03 06:15:16Z
By B+R UnitTest Helper Version: 2.0.1.59
*/
UNITTEST_FIXTURES(fixtures)
{
	new_TestFixture("BrbXXX", BrbXXX),
};

UNITTEST_CALLER_COMPLETE_EXPLICIT(Set_BrbTemplateFunc, "Set_BrbTemplateFunc", 0, 0, fixtures, 0, 0, 0);
```

### Package Logical/UnitTests/UtBrbLibUa - UnitTests for BrbLib

### UnitTest_NoLint.txt
```
Verwendete NOLINTS im Projekt
Diese Angaben sind nur als Hilfe für den ClangTidy-Prüfer des Projekts gedacht und für den Anwender nicht interessant.

BrbLibUa: 136 Stellen
(readability-*, bugprone-easily-swappable-parameters, bugprone-branch-clone, clang-diagnostic-invalid-utf8, clang-diagnostic-invalid-source-encoding, clang-diagnostic-pointer-arith, clang-diagnostic-strict-prototypes, hicpp-uppercase-literal-suffix, cppcoreguidelines-*, performance-*)

UnitTests: 81 Stellen
(readability-*, bugprone-easily-swappable-parameters, bugprone-branch-clone, clang-diagnostic-invalid-utf8, clang-diagnostic-invalid-source-encoding, clang-diagnostic-pointer-arith, clang-diagnostic-strict-prototypes, clang-diagnostic-bad-function-cast, clang-analyzer-security.insecureAPI.*, hicpp-uppercase-literal-suffix, cppcoreguidelines-*, performance-*)

Tasks: 28 Stellen
(readability-*, bugprone-easily-swappable-parameters, bugprone-branch-clone, clang-diagnostic-invalid-utf8, clang-diagnostic-invalid-source-encoding, clang-diagnostic-pointer-arith, clang-diagnostic-strict-prototypes, clang-diagnostic-shadow, clang-diagnostic-bad-function-cast, clang-analyzer-security.insecureAPI.*, hicpp-uppercase-literal-suffix, hicpp-function-size, cppcoreguidelines-*, performance-*)

NOLINT-Kommentare
	// NOLINT()
// NOLINTBEGIN()
// NOLINTEND()
```

### Program Logical/UnitTests/UtBrbLibUa/UtBrbUaStatus (ANSIC) - UnitTests

#### variables.var - Name the suite and add PVs for the program
```iecst
(********************************************************************
 * COPYRIGHT --
 ********************************************************************
 * Program: utTemplate_automated
 * File: variables.var
 * Author: -
 * Created: -
 ********************************************************************
 * Local variables of program utTemplate_automated
 ********************************************************************)
(*Describe the test*)
VAR
	Testsuite : UtMgrTestSuite := (Name:='BrbUaStatus',Description:='(Optional field)Template for use with helper tool. Reference or add this program in the package "TS_UnitTest_UpdateTestPrograms"',Type:=utMgrTEST_TYPE_C,MetaInformation:='(Optional field):To be filled');
END_VAR
(*Input variables for testing*)
VAR
	statusCodeIn0 : UDINT;
	stringIn0 : STRING[256] := '';
END_VAR
(*Functionblock instances for testing*)
(*Output variables for testing*)
VAR
	dwordOut : DWORD;
END_VAR
```

#### autoGeneratedFile.c - Auto generated code - list of all test sets in the program
```c
/*
B+R UnitTest: This is generated code.
Do not edit! Do not move!
Description: UnitTest Testprogramm infrastructure (List of TestSets).
LastUpdated: 2023-04-20 07:17:38Z
By B+R UnitTest Helper Version: 2.0.1.59
*/
#include "UnitTest.h"

UNITTEST_TESTSET_DECLARATION  Set_BrbUaGetStatusCodeText;

UNITTEST_TESTSET_FIXTURES(utTestSets)
{
	new_TestSet(Set_BrbUaGetStatusCodeText),
};
UNTITTEST_TESTSET_HANDLER();
```

#### Set_BrbUaGetStatusCodeText.c - Test set
```c
#include <bur/plctypes.h>

#ifdef _DEFAULT_INCLUDES
#include <AsDefault.h>
#endif

#include "UnitTest.h"
#include "BrbAsserts.h"
#include <string.h>

// NOLINTBEGIN(readability-*, bugprone-easily-swappable-parameters, bugprone-branch-clone, clang-diagnostic-invalid-utf8, clang-diagnostic-invalid-source-encoding, clang-diagnostic-pointer-arith, clang-diagnostic-strict-prototypes, clang-diagnostic-bad-function-cast, clang-analyzer-security.insecureAPI.*, hicpp-uppercase-literal-suffix, cppcoreguidelines-*, performance-*)
_TEST BrbUaGetStatusCodeText_NulPtr(void)
{
	statusCodeIn0 = 0x00000000;
	memset(&stringIn0, 0, sizeof(stringIn0));
	dwordOut = BrbUaGetStatusCodeText(statusCodeIn0, 0, sizeof(stringIn0));
	TEST_ASSERT_EQUAL_INT(0x80460000, dwordOut); // = Bad_StructureMissing
	TEST_ASSERT_EQUAL_STRING("", stringIn0);

	// Finished
	TEST_DONE;
}

_TEST BrbUaGetStatusCodeText_Status(void)
{
	statusCodeIn0 = 0x00000000;
	dwordOut = BrbUaGetStatusCodeText(statusCodeIn0, stringIn0, sizeof(stringIn0));
	TEST_ASSERT_EQUAL_INT(0x00000000, dwordOut); // = Good
	TEST_ASSERT_EQUAL_STRING("0x00000000 = Good", stringIn0);

	statusCodeIn0 = 0xFFFFFFFF;
	dwordOut = BrbUaGetStatusCodeText(statusCodeIn0, stringIn0, sizeof(stringIn0));
	TEST_ASSERT_EQUAL_INT(0x803D0000, dwordOut); // = Bad_NotSupported
	TEST_ASSERT_EQUAL_STRING("0xFFFFFFFF", stringIn0);

	// Finished
	TEST_DONE;
}

// NOLINTEND(readability-*, bugprone-easily-swappable-parameters, bugprone-branch-clone, clang-diagnostic-invalid-utf8, clang-diagnostic-invalid-source-encoding, clang-diagnostic-pointer-arith, clang-diagnostic-strict-prototypes, clang-diagnostic-bad-function-cast, clang-analyzer-security.insecureAPI.*, hicpp-uppercase-literal-suffix, cppcoreguidelines-*, performance-*)

/*
B+R UnitTest: This is generated code.
Do not edit! Do not move!
Description: UnitTest Testprogramm infrastructure (TestSet).
LastUpdated: 2023-04-20 07:23:16Z
By B+R UnitTest Helper Version: 2.0.1.59
*/
UNITTEST_FIXTURES(fixtures)
{
	new_TestFixture("BrbUaGetStatusCodeText_NulPtr", BrbUaGetStatusCodeText_NulPtr),
	new_TestFixture("BrbUaGetStatusCodeText_Status", BrbUaGetStatusCodeText_Status),
};

UNITTEST_CALLER_COMPLETE_EXPLICIT(Set_BrbUaGetStatusCodeText, "Set_BrbUaGetStatusCodeText", 0, 0, fixtures, 0, 0, 0);
```

### Program Logical/UnitTests/UtBrbLibUa/UtBrbUaNodes (ANSIC) - UnitTests

#### variables.var - Name the suite and add PVs for the program
```iecst
(********************************************************************
 * COPYRIGHT --
 ********************************************************************
 * Program: utTemplate_automated
 * File: variables.var
 * Author: -
 * Created: -
 ********************************************************************
 * Local variables of program utTemplate_automated
 ********************************************************************)
(*Describe the test*)
VAR
	Testsuite : UtMgrTestSuite := (Name:='BrbUaNodes',Description:='(Optional field)Template for use with helper tool. Reference or add this program in the package "TS_UnitTest_UpdateTestPrograms"',Type:=utMgrTEST_TYPE_C,MetaInformation:='(Optional field):To be filled');
END_VAR
(*Input variables for testing*)
VAR
	nodeIdIn0 : UANodeID;
	nodeIdIn1 : UANodeID;
	stringIn0 : STRING[256] := '';
	uintIn0 : UINT;
	udintIn0 : UDINT;
END_VAR
(*Functionblock instances for testing*)
(*Output variables for testing*)
VAR
	dwordOut : DWORD;
	boolOut : BOOL;
END_VAR
```

#### autoGeneratedFile.c - Auto generated code - list of all test sets in the program
```c
/*
B+R UnitTest: This is generated code.
Do not edit! Do not move!
Description: UnitTest Testprogramm infrastructure (List of TestSets).
LastUpdated: 2023-04-20 08:30:07Z
By B+R UnitTest Helper Version: 2.0.1.59
*/
#include "UnitTest.h"

UNITTEST_TESTSET_DECLARATION  Set_BrbUaSetNodeId;
UNITTEST_TESTSET_DECLARATION  Set_BrbUaSetNodeIdNum;
UNITTEST_TESTSET_DECLARATION  Set_BrbUaGetRandomNodeId;
UNITTEST_TESTSET_DECLARATION  Set_BrbUaAreNodeIdsEqual;
UNITTEST_TESTSET_DECLARATION  Set_BrbUaAddNodeIdText;

UNITTEST_TESTSET_FIXTURES(utTestSets)
{
	new_TestSet(Set_BrbUaSetNodeId),
	new_TestSet(Set_BrbUaSetNodeIdNum),
	new_TestSet(Set_BrbUaGetRandomNodeId),
	new_TestSet(Set_BrbUaAreNodeIdsEqual),
	new_TestSet(Set_BrbUaAddNodeIdText),
};
UNTITTEST_TESTSET_HANDLER();
```

#### Set_BrbUaSetNodeId.c - Test set
```c
#include <bur/plctypes.h>

#ifdef _DEFAULT_INCLUDES
#include <AsDefault.h>
#endif

#include "UnitTest.h"
#include "BrbAsserts.h"
#include <string.h>

// NOLINTBEGIN(readability-*, bugprone-easily-swappable-parameters, bugprone-branch-clone, clang-diagnostic-invalid-utf8, clang-diagnostic-invalid-source-encoding, clang-diagnostic-pointer-arith, clang-diagnostic-strict-prototypes, clang-diagnostic-bad-function-cast, clang-analyzer-security.insecureAPI.*, hicpp-uppercase-literal-suffix, cppcoreguidelines-*, performance-*)

_TEST BrbUaSetNodeId_NulPtr(void)
{
	memset(&stringIn0, 0, sizeof(stringIn0));
	uintIn0 = 0;
	dwordOut = BrbUaSetNodeId(0, stringIn0, uintIn0);
	TEST_ASSERT_EQUAL_INT(0x80460000, dwordOut); // = Bad_StructureMissing

	// Finished
	TEST_DONE;
}

_TEST BrbUaSetNodeId_Set(void)
{
	strcpy(stringIn0, "VarX");
	uintIn0 = 1;
	dwordOut = BrbUaSetNodeId(&nodeIdIn0, stringIn0, uintIn0);
	TEST_ASSERT_EQUAL_INT(0x00000000, dwordOut); // = Good
	TEST_ASSERT_EQUAL_INT(UAIdentifierType_String, nodeIdIn0.IdentifierType);
	TEST_ASSERT_EQUAL_STRING(stringIn0, nodeIdIn0.Identifier);
	TEST_ASSERT_EQUAL_INT(uintIn0, nodeIdIn0.NamespaceIndex);

	strcpy(stringIn0, "1234");
	uintIn0 = 1;
	dwordOut = BrbUaSetNodeId(&nodeIdIn0, stringIn0, uintIn0);
	TEST_ASSERT_EQUAL_INT(0x00000000, dwordOut); // = Good
	TEST_ASSERT_EQUAL_INT(UAIdentifierType_Numeric, nodeIdIn0.IdentifierType);
	TEST_ASSERT_EQUAL_STRING(stringIn0, nodeIdIn0.Identifier);
	TEST_ASSERT_EQUAL_INT(uintIn0, nodeIdIn0.NamespaceIndex);

	// Finished
	TEST_DONE;
}

// NOLINTEND(readability-*, bugprone-easily-swappable-parameters, bugprone-branch-clone, clang-diagnostic-invalid-utf8, clang-diagnostic-invalid-source-encoding, clang-diagnostic-pointer-arith, clang-diagnostic-strict-prototypes, clang-diagnostic-bad-function-cast, clang-analyzer-security.insecureAPI.*, hicpp-uppercase-literal-suffix, cppcoreguidelines-*, performance-*)

/*
B+R UnitTest: This is generated code.
Do not edit! Do not move!
Description: UnitTest Testprogramm infrastructure (TestSet).
LastUpdated: 2023-04-20 08:00:09Z
By B+R UnitTest Helper Version: 2.0.1.59
*/
UNITTEST_FIXTURES(fixtures)
{
	new_TestFixture("BrbUaSetNodeId_NulPtr", BrbUaSetNodeId_NulPtr),
	new_TestFixture("BrbUaSetNodeId_Set", BrbUaSetNodeId_Set),
};

UNITTEST_CALLER_COMPLETE_EXPLICIT(Set_BrbUaSetNodeId, "Set_BrbUaSetNodeId", 0, 0, fixtures, 0, 0, 0);
```

#### Set_BrbUaSetNodeIdNum.c - Test set
```c
#include <bur/plctypes.h>

#ifdef _DEFAULT_INCLUDES
#include <AsDefault.h>
#endif

#include "UnitTest.h"
#include "BrbAsserts.h"
#include <string.h>

// NOLINTBEGIN(readability-*, bugprone-easily-swappable-parameters, bugprone-branch-clone, clang-diagnostic-invalid-utf8, clang-diagnostic-invalid-source-encoding, clang-diagnostic-pointer-arith, clang-diagnostic-strict-prototypes, clang-diagnostic-bad-function-cast, clang-analyzer-security.insecureAPI.*, hicpp-uppercase-literal-suffix, cppcoreguidelines-*, performance-*)

_TEST BrbUaSetNodeIdNum_NulPtr(void)
{
	udintIn0 = 0;
	uintIn0 = 0;
	dwordOut = BrbUaSetNodeIdNum(0, udintIn0, uintIn0);
	TEST_ASSERT_EQUAL_INT(0x80460000, dwordOut); // = Bad_StructureMissing

	// Finished
	TEST_DONE;
}

_TEST BrbUaSetNodeId_Set(void)
{
	udintIn0 = 1234;
	uintIn0 = 1;
	dwordOut = BrbUaSetNodeIdNum(&nodeIdIn0, udintIn0, uintIn0);
	TEST_ASSERT_EQUAL_INT(0x00000000, dwordOut); // = Good
	TEST_ASSERT_EQUAL_INT(UAIdentifierType_Numeric, nodeIdIn0.IdentifierType);
	TEST_ASSERT_EQUAL_STRING("1234", nodeIdIn0.Identifier);
	TEST_ASSERT_EQUAL_INT(uintIn0, nodeIdIn0.NamespaceIndex);

	// Finished
	TEST_DONE;
}

// NOLINTEND(readability-*, bugprone-easily-swappable-parameters, bugprone-branch-clone, clang-diagnostic-invalid-utf8, clang-diagnostic-invalid-source-encoding, clang-diagnostic-pointer-arith, clang-diagnostic-strict-prototypes, clang-diagnostic-bad-function-cast, clang-analyzer-security.insecureAPI.*, hicpp-uppercase-literal-suffix, cppcoreguidelines-*, performance-*)

/*
B+R UnitTest: This is generated code.
Do not edit! Do not move!
Description: UnitTest Testprogramm infrastructure (TestSet).
LastUpdated: 2023-04-20 08:08:20Z
By B+R UnitTest Helper Version: 2.0.1.59
*/
UNITTEST_FIXTURES(fixtures)
{
	new_TestFixture("BrbUaSetNodeIdNum_NulPtr", BrbUaSetNodeIdNum_NulPtr),
	new_TestFixture("BrbUaSetNodeId_Set", BrbUaSetNodeId_Set),
};

UNITTEST_CALLER_COMPLETE_EXPLICIT(Set_BrbUaSetNodeIdNum, "Set_BrbUaSetNodeIdNum", 0, 0, fixtures, 0, 0, 0);
```

#### Set_BrbUaGetRandomNodeId.c - Test set
```c
#include <bur/plctypes.h>

#ifdef _DEFAULT_INCLUDES
#include <AsDefault.h>
#endif

#include "UnitTest.h"
#include "BrbAsserts.h"
#include <string.h>

// NOLINTBEGIN(readability-*, bugprone-easily-swappable-parameters, bugprone-branch-clone, clang-diagnostic-invalid-utf8, clang-diagnostic-invalid-source-encoding, clang-diagnostic-pointer-arith, clang-diagnostic-strict-prototypes, clang-diagnostic-bad-function-cast, clang-analyzer-security.insecureAPI.*, hicpp-uppercase-literal-suffix, cppcoreguidelines-*, performance-*)

_TEST BrbUaGetRandomNodeId_NulPtr(void)
{
	udintIn0 = 0;
	uintIn0 = 0;
	dwordOut = BrbUaGetRandomNodeId(0, UAIdentifierType_Numeric);
	TEST_ASSERT_EQUAL_INT(0x80460000, dwordOut); // = Bad_StructureMissing

	// Finished
	TEST_DONE;
}

_TEST BrbUaGetRandomNodeId_Get(void)
{
	dwordOut = BrbUaGetRandomNodeId(&nodeIdIn0, UAIdentifierType_Numeric);
	TEST_ASSERT_EQUAL_INT(0x00000000, dwordOut); // = Good
	TEST_ASSERT_EQUAL_INT(UAIdentifierType_Numeric, nodeIdIn0.IdentifierType);

	dwordOut = BrbUaGetRandomNodeId(&nodeIdIn0, UAIdentifierType_String);
	TEST_ASSERT_EQUAL_INT(0x00000000, dwordOut); // = Good
	TEST_ASSERT_EQUAL_INT(UAIdentifierType_String, nodeIdIn0.IdentifierType);

	dwordOut = BrbUaGetRandomNodeId(&nodeIdIn0, UAIdentifierType_GUID);
	TEST_ASSERT_EQUAL_INT(0x00000000, dwordOut); // = Good
	TEST_ASSERT_EQUAL_INT(UAIdentifierType_GUID, nodeIdIn0.IdentifierType);

	dwordOut = BrbUaGetRandomNodeId(&nodeIdIn0, UAIdentifierType_Opaque);
	TEST_ASSERT_EQUAL_INT(0x803D0000, dwordOut); // = Bad_NotSupported
	TEST_ASSERT_EQUAL_INT(UAIdentifierType_Opaque, nodeIdIn0.IdentifierType);

	// Finished
	TEST_DONE;
}

// NOLINTEND(readability-*, bugprone-easily-swappable-parameters, bugprone-branch-clone, clang-diagnostic-invalid-utf8, clang-diagnostic-invalid-source-encoding, clang-diagnostic-pointer-arith, clang-diagnostic-strict-prototypes, clang-diagnostic-bad-function-cast, clang-analyzer-security.insecureAPI.*, hicpp-uppercase-literal-suffix, cppcoreguidelines-*, performance-*)

/*
B+R UnitTest: This is generated code.
Do not edit! Do not move!
Description: UnitTest Testprogramm infrastructure (TestSet).
LastUpdated: 2023-04-20 08:12:57Z
By B+R UnitTest Helper Version: 2.0.1.59
*/
UNITTEST_FIXTURES(fixtures)
{
	new_TestFixture("BrbUaGetRandomNodeId_NulPtr", BrbUaGetRandomNodeId_NulPtr),
	new_TestFixture("BrbUaGetRandomNodeId_Get", BrbUaGetRandomNodeId_Get),
};

UNITTEST_CALLER_COMPLETE_EXPLICIT(Set_BrbUaGetRandomNodeId, "Set_BrbUaGetRandomNodeId", 0, 0, fixtures, 0, 0, 0);
```

#### Set_BrbUaAreNodeIdsEqual.c - Test set
```c
#include <bur/plctypes.h>

#ifdef _DEFAULT_INCLUDES
#include <AsDefault.h>
#endif

#include "UnitTest.h"
#include "BrbAsserts.h"
#include <string.h>

// NOLINTBEGIN(readability-*, bugprone-easily-swappable-parameters, bugprone-branch-clone, clang-diagnostic-invalid-utf8, clang-diagnostic-invalid-source-encoding, clang-diagnostic-pointer-arith, clang-diagnostic-strict-prototypes, clang-diagnostic-bad-function-cast, clang-analyzer-security.insecureAPI.*, hicpp-uppercase-literal-suffix, cppcoreguidelines-*, performance-*)

_TEST BrbUaAreNodeIdsEqual_NulPtr(void)
{
	boolOut = BrbUaAreNodeIdsEqual(0, &nodeIdIn1);
	BRB_ASSERT_EQUAL_BOOL(0, boolOut);

	boolOut = BrbUaAreNodeIdsEqual(&nodeIdIn0, 0);
	BRB_ASSERT_EQUAL_BOOL(0, boolOut);

	// Finished
	TEST_DONE;
}

_TEST BrbUaAreNodeIdsEqual_Compare(void)
{

	BrbUaSetNodeId(&nodeIdIn0, "1234", 12);
	BrbUaSetNodeId(&nodeIdIn1, "1234", 12);
	boolOut = BrbUaAreNodeIdsEqual(&nodeIdIn0, &nodeIdIn1);
	BRB_ASSERT_EQUAL_BOOL(1, boolOut);

	BrbUaSetNodeId(&nodeIdIn0, "1234", 12);
	BrbUaSetNodeId(&nodeIdIn1, "1234", 16);
	boolOut = BrbUaAreNodeIdsEqual(&nodeIdIn0, &nodeIdIn1);
	BRB_ASSERT_EQUAL_BOOL(0, boolOut);

	BrbUaSetNodeId(&nodeIdIn0, "1234", 12);
	BrbUaSetNodeId(&nodeIdIn1, "1235", 12);
	boolOut = BrbUaAreNodeIdsEqual(&nodeIdIn0, &nodeIdIn1);
	BRB_ASSERT_EQUAL_BOOL(0, boolOut);

	BrbUaSetNodeId(&nodeIdIn0, "1234", 12);
	BrbUaSetNodeId(&nodeIdIn1, "1235", 16);
	boolOut = BrbUaAreNodeIdsEqual(&nodeIdIn0, &nodeIdIn1);
	BRB_ASSERT_EQUAL_BOOL(0, boolOut);

	// Finished
	TEST_DONE;
}

// NOLINTEND(readability-*, bugprone-easily-swappable-parameters, bugprone-branch-clone, clang-diagnostic-invalid-utf8, clang-diagnostic-invalid-source-encoding, clang-diagnostic-pointer-arith, clang-diagnostic-strict-prototypes, clang-diagnostic-bad-function-cast, clang-analyzer-security.insecureAPI.*, hicpp-uppercase-literal-suffix, cppcoreguidelines-*, performance-*)

/*
B+R UnitTest: This is generated code.
Do not edit! Do not move!
Description: UnitTest Testprogramm infrastructure (TestSet).
LastUpdated: 2023-04-20 08:16:35Z
By B+R UnitTest Helper Version: 2.0.1.59
*/
UNITTEST_FIXTURES(fixtures)
{
	new_TestFixture("BrbUaAreNodeIdsEqual_NulPtr", BrbUaAreNodeIdsEqual_NulPtr),
	new_TestFixture("BrbUaAreNodeIdsEqual_Compare", BrbUaAreNodeIdsEqual_Compare),
};

UNITTEST_CALLER_COMPLETE_EXPLICIT(Set_BrbUaAreNodeIdsEqual, "Set_BrbUaAreNodeIdsEqual", 0, 0, fixtures, 0, 0, 0);
```

#### Set_BrbUaAddNodeIdText.c - Test set
```c
#include <bur/plctypes.h>

#ifdef _DEFAULT_INCLUDES
#include <AsDefault.h>
#endif

#include "UnitTest.h"
#include "BrbAsserts.h"
#include <string.h>

// NOLINTBEGIN(readability-*, bugprone-easily-swappable-parameters, bugprone-branch-clone, clang-diagnostic-invalid-utf8, clang-diagnostic-invalid-source-encoding, clang-diagnostic-pointer-arith, clang-diagnostic-strict-prototypes, clang-diagnostic-bad-function-cast, clang-analyzer-security.insecureAPI.*, hicpp-uppercase-literal-suffix, cppcoreguidelines-*, performance-*)

_TEST BrbUaAddNodeIdText_NulPtr(void)
{
	dwordOut = BrbUaAddNodeIdText(0, stringIn0, sizeof(stringIn0));
	TEST_ASSERT_EQUAL_INT(0x80460000, dwordOut); // = Bad_StructureMissing

	dwordOut = BrbUaAddNodeIdText(&nodeIdIn0, 0, sizeof(stringIn0));
	TEST_ASSERT_EQUAL_INT(0x80460000, dwordOut); // = Bad_StructureMissing

	// Finished
	TEST_DONE;
}

_TEST BrbUaAddNodeIdText_Add(void)
{
	strcpy(stringIn0, "Test ");
	BrbUaSetNodeId(&nodeIdIn0, "1234", 0);
	dwordOut = BrbUaAddNodeIdText(&nodeIdIn0, stringIn0, sizeof(stringIn0));
	TEST_ASSERT_EQUAL_INT(0x00000000, dwordOut); // = Good
	TEST_ASSERT_EQUAL_STRING("Test ns=0;i=1234", stringIn0);

	strcpy(stringIn0, "Test ");
	BrbUaSetNodeId(&nodeIdIn0, "VarX", 12);
	dwordOut = BrbUaAddNodeIdText(&nodeIdIn0, stringIn0, sizeof(stringIn0));
	TEST_ASSERT_EQUAL_INT(0x00000000, dwordOut); // = Good
	TEST_ASSERT_EQUAL_STRING("Test ns=12;s=VarX", stringIn0);

	strcpy(stringIn0, "Test ");
	nodeIdIn0.IdentifierType = UAIdentifierType_GUID;
	strcpy(nodeIdIn0.Identifier, "12345678-1234-5678-9ABC-123456789ABC");
	nodeIdIn0.NamespaceIndex = 4;
	dwordOut = BrbUaAddNodeIdText(&nodeIdIn0, stringIn0, sizeof(stringIn0));
	TEST_ASSERT_EQUAL_INT(0x00000000, dwordOut); // = Good
	TEST_ASSERT_EQUAL_STRING("Test ns=4;g=12345678-1234-5678-9ABC-123456789ABC", stringIn0);

	strcpy(stringIn0, "Test ");
	nodeIdIn0.IdentifierType = UAIdentifierType_Opaque;
	strcpy(nodeIdIn0.Identifier, "123456789ABCDEF01234");
	nodeIdIn0.NamespaceIndex = 6;
	dwordOut = BrbUaAddNodeIdText(&nodeIdIn0, stringIn0, sizeof(stringIn0));
	TEST_ASSERT_EQUAL_INT(0x00000000, dwordOut); // = Good
	TEST_ASSERT_EQUAL_STRING("Test ns=6;o=123456789ABCDEF01234", stringIn0);

	strcpy(stringIn0, "Test ");
	nodeIdIn0.IdentifierType = 0; // NOLINT(clang-diagnostic-assign-enum)
	strcpy(nodeIdIn0.Identifier, "UnknownIdentifierType");
	nodeIdIn0.NamespaceIndex = 8;
	dwordOut = BrbUaAddNodeIdText(&nodeIdIn0, stringIn0, sizeof(stringIn0));
	TEST_ASSERT_EQUAL_INT(0x00000000, dwordOut); // = Good
	TEST_ASSERT_EQUAL_STRING("Test ns=8;?=UnknownIdentifierType", stringIn0);

	// Finished
	TEST_DONE;
}

// NOLINTEND(readability-*, bugprone-easily-swappable-parameters, bugprone-branch-clone, clang-diagnostic-invalid-utf8, clang-diagnostic-invalid-source-encoding, clang-diagnostic-pointer-arith, clang-diagnostic-strict-prototypes, clang-diagnostic-bad-function-cast, clang-analyzer-security.insecureAPI.*, hicpp-uppercase-literal-suffix, cppcoreguidelines-*, performance-*)

/*
B+R UnitTest: This is generated code.
Do not edit! Do not move!
Description: UnitTest Testprogramm infrastructure (TestSet).
LastUpdated: 2023-04-20 08:30:07Z
By B+R UnitTest Helper Version: 2.0.1.59
*/
UNITTEST_FIXTURES(fixtures)
{
	new_TestFixture("BrbUaAddNodeIdText_NulPtr", BrbUaAddNodeIdText_NulPtr),
	new_TestFixture("BrbUaAddNodeIdText_Add", BrbUaAddNodeIdText_Add),
};

UNITTEST_CALLER_COMPLETE_EXPLICIT(Set_BrbUaAddNodeIdText, "Set_BrbUaAddNodeIdText", 0, 0, fixtures, 0, 0, 0);
```

### Program Logical/UnitTests/UtBrbLibUa/UtBrbUaAttributes (ANSIC) - UnitTests

#### variables.var - Name the suite and add PVs for the program
```iecst
(********************************************************************
 * COPYRIGHT --
 ********************************************************************
 * Program: utTemplate_automated
 * File: variables.var
 * Author: -
 * Created: -
 ********************************************************************
 * Local variables of program utTemplate_automated
 ********************************************************************)
(*Describe the test*)
VAR
	Testsuite : UtMgrTestSuite := (Name:='BrbUaAttributes',Description:='(Optional field)Template for use with helper tool. Reference or add this program in the package "TS_UnitTest_UpdateTestPrograms"',Type:=utMgrTEST_TYPE_C,MetaInformation:='(Optional field):To be filled');
END_VAR
(*Constants*)
VAR CONSTANT
	nARRAY_DIMENSION_INDEX_MAX : UINT := 5;
END_VAR
(*Input variables for testing*)
VAR
	stringIn0 : STRING[256] := '';
	anArrayDimensions : ARRAY[0..nARRAY_DIMENSION_INDEX_MAX] OF UDINT;
END_VAR
(*Functionblock instances for testing*)
(*Output variables for testing*)
VAR
	dwordOut : DWORD;
	varianTypeOut : UAVariantType;
END_VAR
```

#### autoGeneratedFile.c - Auto generated code - list of all test sets in the program
```c
/*
B+R UnitTest: This is generated code.
Do not edit! Do not move!
Description: UnitTest Testprogramm infrastructure (List of TestSets).
LastUpdated: 2023-04-20 09:47:06Z
By B+R UnitTest Helper Version: 2.0.1.59
*/
#include "UnitTest.h"

UNITTEST_TESTSET_DECLARATION  Set_BrbUaGetAttributeIdDatatype;
UNITTEST_TESTSET_DECLARATION  Set_BrbUaAddBooleanText;
UNITTEST_TESTSET_DECLARATION  Set_BrbUaAddNodeClassText;
UNITTEST_TESTSET_DECLARATION  Set_BrbUaAddDatatypeIdText;
UNITTEST_TESTSET_DECLARATION  Set_BrbUaAddArrayDimensionText;
UNITTEST_TESTSET_DECLARATION  Set_BrbUaAddAccessLevelText;
UNITTEST_TESTSET_DECLARATION  Set_BrbUaAddEventNotifierText;

UNITTEST_TESTSET_FIXTURES(utTestSets)
{
	new_TestSet(Set_BrbUaGetAttributeIdDatatype),
	new_TestSet(Set_BrbUaAddBooleanText),
	new_TestSet(Set_BrbUaAddNodeClassText),
	new_TestSet(Set_BrbUaAddDatatypeIdText),
	new_TestSet(Set_BrbUaAddArrayDimensionText),
	new_TestSet(Set_BrbUaAddAccessLevelText),
	new_TestSet(Set_BrbUaAddEventNotifierText),
};
UNTITTEST_TESTSET_HANDLER();
```

#### Set_BrbUaGetAttributeIdDatatype.c - Test set
```c
#include <bur/plctypes.h>

#ifdef _DEFAULT_INCLUDES
#include <AsDefault.h>
#endif

#include "UnitTest.h"
#include "BrbAsserts.h"
#include <string.h>

// NOLINTBEGIN(readability-*, bugprone-easily-swappable-parameters, bugprone-branch-clone, clang-diagnostic-invalid-utf8, clang-diagnostic-invalid-source-encoding, clang-diagnostic-pointer-arith, clang-diagnostic-strict-prototypes, clang-diagnostic-bad-function-cast, clang-analyzer-security.insecureAPI.*, hicpp-uppercase-literal-suffix, cppcoreguidelines-*, performance-*)

_TEST BrbUaGetAttributeIdDatatype_Get(void)
{

	varianTypeOut = BrbUaGetAttributeIdDatatype(UAAI_Default);
	BRB_ASSERT_EQUAL_DINT(UAVariantType_Null, (DINT)varianTypeOut);

	varianTypeOut = BrbUaGetAttributeIdDatatype(UAAI_NodeId);
	BRB_ASSERT_EQUAL_DINT(UAVariantType_NodeId, (DINT)varianTypeOut);

	varianTypeOut = BrbUaGetAttributeIdDatatype(UAAI_UserExecutable);
	BRB_ASSERT_EQUAL_DINT(UAVariantType_Boolean, (DINT)varianTypeOut);

	// Finished
	TEST_DONE;
}

// NOLINTEND(readability-*, bugprone-easily-swappable-parameters, bugprone-branch-clone, clang-diagnostic-invalid-utf8, clang-diagnostic-invalid-source-encoding, clang-diagnostic-pointer-arith, clang-diagnostic-strict-prototypes, clang-diagnostic-bad-function-cast, clang-analyzer-security.insecureAPI.*, hicpp-uppercase-literal-suffix, cppcoreguidelines-*, performance-*)

/*
B+R UnitTest: This is generated code.
Do not edit! Do not move!
Description: UnitTest Testprogramm infrastructure (TestSet).
LastUpdated: 2023-04-20 08:53:32Z
By B+R UnitTest Helper Version: 2.0.1.59
*/
UNITTEST_FIXTURES(fixtures)
{
	new_TestFixture("BrbUaGetAttributeIdDatatype_Get", BrbUaGetAttributeIdDatatype_Get),
};

UNITTEST_CALLER_COMPLETE_EXPLICIT(Set_BrbUaGetAttributeIdDatatype, "Set_BrbUaGetAttributeIdDatatype", 0, 0, fixtures, 0, 0, 0);
```

#### Set_BrbUaAddBooleanText.c - Test set
```c
#include <bur/plctypes.h>

#ifdef _DEFAULT_INCLUDES
#include <AsDefault.h>
#endif

#include "UnitTest.h"
#include "BrbAsserts.h"
#include <string.h>

// NOLINTBEGIN(readability-*, bugprone-easily-swappable-parameters, bugprone-branch-clone, clang-diagnostic-invalid-utf8, clang-diagnostic-invalid-source-encoding, clang-diagnostic-pointer-arith, clang-diagnostic-strict-prototypes, clang-diagnostic-bad-function-cast, clang-analyzer-security.insecureAPI.*, hicpp-uppercase-literal-suffix, cppcoreguidelines-*, performance-*)

_TEST BrbUaAddBooleanText_NulPtr(void)
{
	dwordOut = BrbUaAddBooleanText(0, 0, sizeof(stringIn0));
	TEST_ASSERT_EQUAL_INT(0x80460000, dwordOut); // = Bad_StructureMissing

	// Finished
	TEST_DONE;
}

_TEST BrbUaAddBooleanText_Add(void)
{
	strcpy(stringIn0, "Test ");
	dwordOut = BrbUaAddBooleanText(0, stringIn0, sizeof(stringIn0));
	TEST_ASSERT_EQUAL_INT(0x00000000, dwordOut); // = Good
	TEST_ASSERT_EQUAL_STRING("Test False", stringIn0);

	strcpy(stringIn0, "Test ");
	dwordOut = BrbUaAddBooleanText(1, stringIn0, sizeof(stringIn0));
	TEST_ASSERT_EQUAL_INT(0x00000000, dwordOut); // = Good
	TEST_ASSERT_EQUAL_STRING("Test True", stringIn0);

	// Finished
	TEST_DONE;
}

// NOLINTEND(readability-*, bugprone-easily-swappable-parameters, bugprone-branch-clone, clang-diagnostic-invalid-utf8, clang-diagnostic-invalid-source-encoding, clang-diagnostic-pointer-arith, clang-diagnostic-strict-prototypes, clang-diagnostic-bad-function-cast, clang-analyzer-security.insecureAPI.*, hicpp-uppercase-literal-suffix, cppcoreguidelines-*, performance-*)

/*
B+R UnitTest: This is generated code.
Do not edit! Do not move!
Description: UnitTest Testprogramm infrastructure (TestSet).
LastUpdated: 2023-04-20 08:59:46Z
By B+R UnitTest Helper Version: 2.0.1.59
*/
UNITTEST_FIXTURES(fixtures)
{
	new_TestFixture("BrbUaAddBooleanText_NulPtr", BrbUaAddBooleanText_NulPtr),
	new_TestFixture("BrbUaAddBooleanText_Add", BrbUaAddBooleanText_Add),
};

UNITTEST_CALLER_COMPLETE_EXPLICIT(Set_BrbUaAddBooleanText, "Set_BrbUaAddBooleanText", 0, 0, fixtures, 0, 0, 0);
```

#### Set_BrbUaAddNodeClassText.c - Test set
```c
#include <bur/plctypes.h>

#ifdef _DEFAULT_INCLUDES
#include <AsDefault.h>
#endif

#include "UnitTest.h"
#include "BrbAsserts.h"
#include <string.h>

// NOLINTBEGIN(readability-*, bugprone-easily-swappable-parameters, bugprone-branch-clone, clang-diagnostic-invalid-utf8, clang-diagnostic-invalid-source-encoding, clang-diagnostic-pointer-arith, clang-diagnostic-strict-prototypes, clang-diagnostic-bad-function-cast, clang-analyzer-security.insecureAPI.*, hicpp-uppercase-literal-suffix, cppcoreguidelines-*, performance-*)

_TEST BrbUaAddNodeClassText_NulPtr(void)
{
	dwordOut = BrbUaAddNodeClassText(UANodeClass_None, 0, sizeof(stringIn0));
	TEST_ASSERT_EQUAL_INT(0x80460000, dwordOut); // = Bad_StructureMissing

	// Finished
	TEST_DONE;
}

_TEST BrbUaAddNodeClassText_Add(void)
{
	strcpy(stringIn0, "Test ");
	dwordOut = BrbUaAddNodeClassText(UANodeClass_None, stringIn0, sizeof(stringIn0));
	TEST_ASSERT_EQUAL_INT(0x00000000, dwordOut); // = Good
	TEST_ASSERT_EQUAL_STRING("Test None", stringIn0);

	strcpy(stringIn0, "Test ");
	dwordOut = BrbUaAddNodeClassText(UANodeClass_Object, stringIn0, sizeof(stringIn0));
	TEST_ASSERT_EQUAL_INT(0x00000000, dwordOut); // = Good
	TEST_ASSERT_EQUAL_STRING("Test Object", stringIn0);

	strcpy(stringIn0, "Test ");
	dwordOut = BrbUaAddNodeClassText(UANodeClass_Variable, stringIn0, sizeof(stringIn0));
	TEST_ASSERT_EQUAL_INT(0x00000000, dwordOut); // = Good
	TEST_ASSERT_EQUAL_STRING("Test Variable", stringIn0);

	strcpy(stringIn0, "Test ");
	dwordOut = BrbUaAddNodeClassText(UANodeClass_Method, stringIn0, sizeof(stringIn0));
	TEST_ASSERT_EQUAL_INT(0x00000000, dwordOut); // = Good
	TEST_ASSERT_EQUAL_STRING("Test Method", stringIn0);

	strcpy(stringIn0, "Test ");
	dwordOut = BrbUaAddNodeClassText(254, stringIn0, sizeof(stringIn0)); // NOLINT(clang-diagnostic-assign-enum)
	TEST_ASSERT_EQUAL_INT(0x00000000, dwordOut); // = Good
	TEST_ASSERT_EQUAL_STRING("Test Unknown", stringIn0);

	// Finished
	TEST_DONE;
}

// NOLINTEND(readability-*, bugprone-easily-swappable-parameters, bugprone-branch-clone, clang-diagnostic-invalid-utf8, clang-diagnostic-invalid-source-encoding, clang-diagnostic-pointer-arith, clang-diagnostic-strict-prototypes, clang-diagnostic-bad-function-cast, clang-analyzer-security.insecureAPI.*, hicpp-uppercase-literal-suffix, cppcoreguidelines-*, performance-*)

/*
B+R UnitTest: This is generated code.
Do not edit! Do not move!
Description: UnitTest Testprogramm infrastructure (TestSet).
LastUpdated: 2023-04-20 09:05:44Z
By B+R UnitTest Helper Version: 2.0.1.59
*/
UNITTEST_FIXTURES(fixtures)
{
	new_TestFixture("BrbUaAddNodeClassText_NulPtr", BrbUaAddNodeClassText_NulPtr),
	new_TestFixture("BrbUaAddNodeClassText_Add", BrbUaAddNodeClassText_Add),
};

UNITTEST_CALLER_COMPLETE_EXPLICIT(Set_BrbUaAddNodeClassText, "Set_BrbUaAddNodeClassText", 0, 0, fixtures, 0, 0, 0);
```

#### Set_BrbUaAddDatatypeIdText.c - Test set
```c
#include <bur/plctypes.h>

#ifdef _DEFAULT_INCLUDES
#include <AsDefault.h>
#endif

#include "UnitTest.h"
#include "BrbAsserts.h"
#include <string.h>

// NOLINTBEGIN(readability-*, bugprone-easily-swappable-parameters, bugprone-branch-clone, clang-diagnostic-invalid-utf8, clang-diagnostic-invalid-source-encoding, clang-diagnostic-pointer-arith, clang-diagnostic-strict-prototypes, clang-diagnostic-bad-function-cast, clang-analyzer-security.insecureAPI.*, hicpp-uppercase-literal-suffix, cppcoreguidelines-*, performance-*)

_TEST BrbUaAddDatatypeIdText_NulPtr(void)
{
	dwordOut = BrbUaAddDatatypeIdText(0, 0, sizeof(stringIn0));
	TEST_ASSERT_EQUAL_INT(0x80460000, dwordOut); // = Bad_StructureMissing

	// Finished
	TEST_DONE;
}

_TEST BrbUaAddDatatypeIdText_Add(void)
{
	strcpy(stringIn0, "Test ");
	dwordOut = BrbUaAddDatatypeIdText(1, stringIn0, sizeof(stringIn0));
	TEST_ASSERT_EQUAL_INT(0x00000000, dwordOut); // = Good
	TEST_ASSERT_EQUAL_STRING("Test 1=Boolean", stringIn0);

	strcpy(stringIn0, "Test ");
	dwordOut = BrbUaAddDatatypeIdText(4, stringIn0, sizeof(stringIn0));
	TEST_ASSERT_EQUAL_INT(0x00000000, dwordOut); // = Good
	TEST_ASSERT_EQUAL_STRING("Test 4=Int16", stringIn0);

	strcpy(stringIn0, "Test ");
	dwordOut = BrbUaAddDatatypeIdText(8, stringIn0, sizeof(stringIn0));
	TEST_ASSERT_EQUAL_INT(0x00000000, dwordOut); // = Good
	TEST_ASSERT_EQUAL_STRING("Test 8=Int64", stringIn0);

	strcpy(stringIn0, "Test ");
	dwordOut = BrbUaAddDatatypeIdText(12, stringIn0, sizeof(stringIn0));
	TEST_ASSERT_EQUAL_INT(0x00000000, dwordOut); // = Good
	TEST_ASSERT_EQUAL_STRING("Test 12=String", stringIn0);

	strcpy(stringIn0, "Test ");
	dwordOut = BrbUaAddDatatypeIdText(15, stringIn0, sizeof(stringIn0));
	TEST_ASSERT_EQUAL_INT(0x00000000, dwordOut); // = Good
	TEST_ASSERT_EQUAL_STRING("Test 15=ByteString", stringIn0);

	strcpy(stringIn0, "Test ");
	dwordOut = BrbUaAddDatatypeIdText(17, stringIn0, sizeof(stringIn0));
	TEST_ASSERT_EQUAL_INT(0x00000000, dwordOut); // = Good
	TEST_ASSERT_EQUAL_STRING("Test 17=NodeId", stringIn0);

	strcpy(stringIn0, "Test ");
	dwordOut = BrbUaAddDatatypeIdText(22, stringIn0, sizeof(stringIn0));
	TEST_ASSERT_EQUAL_INT(0x00000000, dwordOut); // = Good
	TEST_ASSERT_EQUAL_STRING("Test 22=Structure", stringIn0);

	strcpy(stringIn0, "Test ");
	dwordOut = BrbUaAddDatatypeIdText(0, stringIn0, sizeof(stringIn0));
	TEST_ASSERT_EQUAL_INT(0x00000000, dwordOut); // = Good
	TEST_ASSERT_EQUAL_STRING("Test 0", stringIn0);

	// Finished
	TEST_DONE;
}

// NOLINTEND(readability-*, bugprone-easily-swappable-parameters, bugprone-branch-clone, clang-diagnostic-invalid-utf8, clang-diagnostic-invalid-source-encoding, clang-diagnostic-pointer-arith, clang-diagnostic-strict-prototypes, clang-diagnostic-bad-function-cast, clang-analyzer-security.insecureAPI.*, hicpp-uppercase-literal-suffix, cppcoreguidelines-*, performance-*)

/*
B+R UnitTest: This is generated code.
Do not edit! Do not move!
Description: UnitTest Testprogramm infrastructure (TestSet).
LastUpdated: 2023-04-20 09:10:48Z
By B+R UnitTest Helper Version: 2.0.1.59
*/
UNITTEST_FIXTURES(fixtures)
{
	new_TestFixture("BrbUaAddDatatypeIdText_NulPtr", BrbUaAddDatatypeIdText_NulPtr),
	new_TestFixture("BrbUaAddDatatypeIdText_Add", BrbUaAddDatatypeIdText_Add),
};

UNITTEST_CALLER_COMPLETE_EXPLICIT(Set_BrbUaAddDatatypeIdText, "Set_BrbUaAddDatatypeIdText", 0, 0, fixtures, 0, 0, 0);
```

#### Set_BrbUaAddArrayDimensionText.c - Test set
```c
#include <bur/plctypes.h>

#ifdef _DEFAULT_INCLUDES
#include <AsDefault.h>
#endif

#include "UnitTest.h"
#include "BrbAsserts.h"
#include <string.h>

// NOLINTBEGIN(readability-*, bugprone-easily-swappable-parameters, bugprone-branch-clone, clang-diagnostic-invalid-utf8, clang-diagnostic-invalid-source-encoding, clang-diagnostic-pointer-arith, clang-diagnostic-strict-prototypes, clang-diagnostic-bad-function-cast, clang-analyzer-security.insecureAPI.*, hicpp-uppercase-literal-suffix, cppcoreguidelines-*, performance-*)

_TEST BrbUaAddArrayDimensionText_NulPtr(void)
{
	dwordOut = BrbUaAddArrayDimensionText(0, nARRAY_DIMENSION_INDEX_MAX, stringIn0, sizeof(stringIn0));
	TEST_ASSERT_EQUAL_INT(0x80460000, dwordOut); // = Bad_StructureMissing

	dwordOut = BrbUaAddArrayDimensionText((UDINT*)&anArrayDimensions, nARRAY_DIMENSION_INDEX_MAX, 0, sizeof(stringIn0));
	TEST_ASSERT_EQUAL_INT(0x80460000, dwordOut); // = Bad_StructureMissing

	// Finished
	TEST_DONE;
}

_TEST BrbUaAddArrayDimensionText_Add(void)
{
	anArrayDimensions[0] = 1;
	anArrayDimensions[1] = 2;
	anArrayDimensions[2] = 3;
	anArrayDimensions[3] = 4;
	anArrayDimensions[4] = 5;
	anArrayDimensions[5] = 6;

	strcpy(stringIn0, "Test ");
	dwordOut = BrbUaAddArrayDimensionText((UDINT*)&anArrayDimensions, 0, stringIn0, sizeof(stringIn0));
	TEST_ASSERT_EQUAL_INT(0x800F0000 , dwordOut); // = Bad_NothingToDo
	TEST_ASSERT_EQUAL_STRING("Test ", stringIn0);

	strcpy(stringIn0, "Test ");
	dwordOut = BrbUaAddArrayDimensionText((UDINT*)&anArrayDimensions, 1, stringIn0, sizeof(stringIn0));
	TEST_ASSERT_EQUAL_INT(0x00000000, dwordOut); // = Good
	TEST_ASSERT_EQUAL_STRING("Test 1", stringIn0);

	strcpy(stringIn0, "Test ");
	dwordOut = BrbUaAddArrayDimensionText((UDINT*)&anArrayDimensions, 3, stringIn0, sizeof(stringIn0));
	TEST_ASSERT_EQUAL_INT(0x00000000, dwordOut); // = Good
	TEST_ASSERT_EQUAL_STRING("Test 1;2;3", stringIn0);

	strcpy(stringIn0, "Test ");
	dwordOut = BrbUaAddArrayDimensionText((UDINT*)&anArrayDimensions, 6, stringIn0, sizeof(stringIn0));
	TEST_ASSERT_EQUAL_INT(0x00000000, dwordOut); // = Good
	TEST_ASSERT_EQUAL_STRING("Test 1;2;3;4;5;6", stringIn0);

	// Finished
	TEST_DONE;
}

// NOLINTEND(readability-*, bugprone-easily-swappable-parameters, bugprone-branch-clone, clang-diagnostic-invalid-utf8, clang-diagnostic-invalid-source-encoding, clang-diagnostic-pointer-arith, clang-diagnostic-strict-prototypes, clang-diagnostic-bad-function-cast, clang-analyzer-security.insecureAPI.*, hicpp-uppercase-literal-suffix, cppcoreguidelines-*, performance-*)

/*
B+R UnitTest: This is generated code.
Do not edit! Do not move!
Description: UnitTest Testprogramm infrastructure (TestSet).
LastUpdated: 2023-04-20 09:18:31Z
By B+R UnitTest Helper Version: 2.0.1.59
*/
UNITTEST_FIXTURES(fixtures)
{
	new_TestFixture("BrbUaAddArrayDimensionText_NulPtr", BrbUaAddArrayDimensionText_NulPtr),
	new_TestFixture("BrbUaAddArrayDimensionText_Add", BrbUaAddArrayDimensionText_Add),
};

UNITTEST_CALLER_COMPLETE_EXPLICIT(Set_BrbUaAddArrayDimensionText, "Set_BrbUaAddArrayDimensionText", 0, 0, fixtures, 0, 0, 0);
```

#### Set_BrbUaAddAccessLevelText.c - Test set
```c
#include <bur/plctypes.h>

#ifdef _DEFAULT_INCLUDES
#include <AsDefault.h>
#endif

#include "UnitTest.h"
#include "BrbAsserts.h"
#include <string.h>

// NOLINTBEGIN(readability-*, bugprone-easily-swappable-parameters, bugprone-branch-clone, clang-diagnostic-invalid-utf8, clang-diagnostic-invalid-source-encoding, clang-diagnostic-pointer-arith, clang-diagnostic-strict-prototypes, clang-diagnostic-bad-function-cast, clang-analyzer-security.insecureAPI.*, hicpp-uppercase-literal-suffix, cppcoreguidelines-*, performance-*)

_TEST BrbUaAddAccessLevelText_NulPtr(void)
{
	dwordOut = BrbUaAddAccessLevelText(0, 0, sizeof(stringIn0));
	TEST_ASSERT_EQUAL_INT(0x80460000, dwordOut); // = Bad_StructureMissing

	// Finished
	TEST_DONE;
}

_TEST BrbUaAddAccessLevelText_Add(void)
{
	strcpy(stringIn0, "Test ");
	dwordOut = BrbUaAddAccessLevelText(0, stringIn0, sizeof(stringIn0));
	TEST_ASSERT_EQUAL_INT(0x00000000, dwordOut); // = Good
	TEST_ASSERT_EQUAL_STRING("Test 0= None", stringIn0);

	strcpy(stringIn0, "Test ");
	dwordOut = BrbUaAddAccessLevelText(1, stringIn0, sizeof(stringIn0));
	TEST_ASSERT_EQUAL_INT(0x00000000, dwordOut); // = Good
	TEST_ASSERT_EQUAL_STRING("Test 1= Read", stringIn0);

	strcpy(stringIn0, "Test ");
	dwordOut = BrbUaAddAccessLevelText(2, stringIn0, sizeof(stringIn0));
	TEST_ASSERT_EQUAL_INT(0x00000000, dwordOut); // = Good
	TEST_ASSERT_EQUAL_STRING("Test 2= Write", stringIn0);

	strcpy(stringIn0, "Test ");
	dwordOut = BrbUaAddAccessLevelText(3, stringIn0, sizeof(stringIn0));
	TEST_ASSERT_EQUAL_INT(0x00000000, dwordOut); // = Good
	TEST_ASSERT_EQUAL_STRING("Test 3= Read, Write", stringIn0);

	strcpy(stringIn0, "Test ");
	dwordOut = BrbUaAddAccessLevelText(4, stringIn0, sizeof(stringIn0));
	TEST_ASSERT_EQUAL_INT(0x00000000, dwordOut); // = Good
	TEST_ASSERT_EQUAL_STRING("Test 4= HistoryRead", stringIn0);

	strcpy(stringIn0, "Test ");
	dwordOut = BrbUaAddAccessLevelText(5, stringIn0, sizeof(stringIn0));
	TEST_ASSERT_EQUAL_INT(0x00000000, dwordOut); // = Good
	TEST_ASSERT_EQUAL_STRING("Test 5= Read, HistoryRead", stringIn0);

	strcpy(stringIn0, "Test ");
	dwordOut = BrbUaAddAccessLevelText(6, stringIn0, sizeof(stringIn0));
	TEST_ASSERT_EQUAL_INT(0x00000000, dwordOut); // = Good
	TEST_ASSERT_EQUAL_STRING("Test 6= Write, HistoryRead", stringIn0);

	strcpy(stringIn0, "Test ");
	dwordOut = BrbUaAddAccessLevelText(7, stringIn0, sizeof(stringIn0));
	TEST_ASSERT_EQUAL_INT(0x00000000, dwordOut); // = Good
	TEST_ASSERT_EQUAL_STRING("Test 7= Read, Write, HistoryRead", stringIn0);

	strcpy(stringIn0, "Test ");
	dwordOut = BrbUaAddAccessLevelText(8, stringIn0, sizeof(stringIn0));
	TEST_ASSERT_EQUAL_INT(0x00000000, dwordOut); // = Good
	TEST_ASSERT_EQUAL_STRING("Test 8= HistoryWrite", stringIn0);

	strcpy(stringIn0, "Test ");
	dwordOut = BrbUaAddAccessLevelText(9, stringIn0, sizeof(stringIn0));
	TEST_ASSERT_EQUAL_INT(0x00000000, dwordOut); // = Good
	TEST_ASSERT_EQUAL_STRING("Test 9= Read, HistoryWrite", stringIn0);

	strcpy(stringIn0, "Test ");
	dwordOut = BrbUaAddAccessLevelText(10, stringIn0, sizeof(stringIn0));
	TEST_ASSERT_EQUAL_INT(0x00000000, dwordOut); // = Good
	TEST_ASSERT_EQUAL_STRING("Test 10= Write, HistoryWrite", stringIn0);

	strcpy(stringIn0, "Test ");
	dwordOut = BrbUaAddAccessLevelText(11, stringIn0, sizeof(stringIn0));
	TEST_ASSERT_EQUAL_INT(0x00000000, dwordOut); // = Good
	TEST_ASSERT_EQUAL_STRING("Test 11= Read, Write, HistoryWrite", stringIn0);

	strcpy(stringIn0, "Test ");
	dwordOut = BrbUaAddAccessLevelText(12, stringIn0, sizeof(stringIn0));
	TEST_ASSERT_EQUAL_INT(0x00000000, dwordOut); // = Good
	TEST_ASSERT_EQUAL_STRING("Test 12= HistoryRead, HistoryWrite", stringIn0);

	strcpy(stringIn0, "Test ");
	dwordOut = BrbUaAddAccessLevelText(13, stringIn0, sizeof(stringIn0));
	TEST_ASSERT_EQUAL_INT(0x00000000, dwordOut); // = Good
	TEST_ASSERT_EQUAL_STRING("Test 13= Read, HistoryRead, HistoryWrite", stringIn0);

	strcpy(stringIn0, "Test ");
	dwordOut = BrbUaAddAccessLevelText(14, stringIn0, sizeof(stringIn0));
	TEST_ASSERT_EQUAL_INT(0x00000000, dwordOut); // = Good
	TEST_ASSERT_EQUAL_STRING("Test 14= Write, HistoryRead, HistoryWrite", stringIn0);

	strcpy(stringIn0, "Test ");
	dwordOut = BrbUaAddAccessLevelText(15, stringIn0, sizeof(stringIn0));
	TEST_ASSERT_EQUAL_INT(0x00000000, dwordOut); // = Good
	TEST_ASSERT_EQUAL_STRING("Test 15= Read, Write, HistoryRead, HistoryWrite", stringIn0);

	// Finished
	TEST_DONE;
}

// NOLINTEND(readability-*, bugprone-easily-swappable-parameters, bugprone-branch-clone, clang-diagnostic-invalid-utf8, clang-diagnostic-invalid-source-encoding, clang-diagnostic-pointer-arith, clang-diagnostic-strict-prototypes, clang-diagnostic-bad-function-cast, clang-analyzer-security.insecureAPI.*, hicpp-uppercase-literal-suffix, cppcoreguidelines-*, performance-*)

/*
B+R UnitTest: This is generated code.
Do not edit! Do not move!
Description: UnitTest Testprogramm infrastructure (TestSet).
LastUpdated: 2023-04-20 09:38:10Z
By B+R UnitTest Helper Version: 2.0.1.59
*/
UNITTEST_FIXTURES(fixtures)
{
	new_TestFixture("BrbUaAddAccessLevelText_NulPtr", BrbUaAddAccessLevelText_NulPtr),
	new_TestFixture("BrbUaAddAccessLevelText_Add", BrbUaAddAccessLevelText_Add),
};

UNITTEST_CALLER_COMPLETE_EXPLICIT(Set_BrbUaAddAccessLevelText, "Set_BrbUaAddAccessLevelText", 0, 0, fixtures, 0, 0, 0);
```

#### Set_BrbUaAddEventNotifierText.c - Test set
```c
#include <bur/plctypes.h>

#ifdef _DEFAULT_INCLUDES
#include <AsDefault.h>
#endif

#include "UnitTest.h"
#include "BrbAsserts.h"
#include <string.h>

// NOLINTBEGIN(readability-*, bugprone-easily-swappable-parameters, bugprone-branch-clone, clang-diagnostic-invalid-utf8, clang-diagnostic-invalid-source-encoding, clang-diagnostic-pointer-arith, clang-diagnostic-strict-prototypes, clang-diagnostic-bad-function-cast, clang-analyzer-security.insecureAPI.*, hicpp-uppercase-literal-suffix, cppcoreguidelines-*, performance-*)

_TEST BrbUaAddEventNotifierText_NulPtr(void)
{
	dwordOut = BrbUaAddEventNotifierText(0, 0, sizeof(stringIn0));
	TEST_ASSERT_EQUAL_INT(0x80460000, dwordOut); // = Bad_StructureMissing

	// Finished
	TEST_DONE;
}

_TEST BrbUaAddEventNotifierText_Add(void)
{
	strcpy(stringIn0, "Test ");
	dwordOut = BrbUaAddEventNotifierText(0, stringIn0, sizeof(stringIn0));
	TEST_ASSERT_EQUAL_INT(0x00000000, dwordOut); // = Good
	TEST_ASSERT_EQUAL_STRING("Test 0= None", stringIn0);

	strcpy(stringIn0, "Test ");
	dwordOut = BrbUaAddEventNotifierText(1, stringIn0, sizeof(stringIn0));
	TEST_ASSERT_EQUAL_INT(0x00000000, dwordOut); // = Good
	TEST_ASSERT_EQUAL_STRING("Test 1= Subscribe", stringIn0);

	strcpy(stringIn0, "Test ");
	dwordOut = BrbUaAddEventNotifierText(2, stringIn0, sizeof(stringIn0));
	TEST_ASSERT_EQUAL_INT(0x00000000, dwordOut); // = Good
	TEST_ASSERT_EQUAL_STRING("Test 2=", stringIn0);

	strcpy(stringIn0, "Test ");
	dwordOut = BrbUaAddEventNotifierText(3, stringIn0, sizeof(stringIn0));
	TEST_ASSERT_EQUAL_INT(0x00000000, dwordOut); // = Good
	TEST_ASSERT_EQUAL_STRING("Test 3= Subscribe", stringIn0);

	strcpy(stringIn0, "Test ");
	dwordOut = BrbUaAddEventNotifierText(4, stringIn0, sizeof(stringIn0));
	TEST_ASSERT_EQUAL_INT(0x00000000, dwordOut); // = Good
	TEST_ASSERT_EQUAL_STRING("Test 4= HistoryRead", stringIn0);

	strcpy(stringIn0, "Test ");
	dwordOut = BrbUaAddEventNotifierText(5, stringIn0, sizeof(stringIn0));
	TEST_ASSERT_EQUAL_INT(0x00000000, dwordOut); // = Good
	TEST_ASSERT_EQUAL_STRING("Test 5= Subscribe, HistoryRead", stringIn0);

	strcpy(stringIn0, "Test ");
	dwordOut = BrbUaAddEventNotifierText(6, stringIn0, sizeof(stringIn0));
	TEST_ASSERT_EQUAL_INT(0x00000000, dwordOut); // = Good
	TEST_ASSERT_EQUAL_STRING("Test 6= HistoryRead", stringIn0);

	strcpy(stringIn0, "Test ");
	dwordOut = BrbUaAddEventNotifierText(7, stringIn0, sizeof(stringIn0));
	TEST_ASSERT_EQUAL_INT(0x00000000, dwordOut); // = Good
	TEST_ASSERT_EQUAL_STRING("Test 7= Subscribe, HistoryRead", stringIn0);

	strcpy(stringIn0, "Test ");
	dwordOut = BrbUaAddEventNotifierText(8, stringIn0, sizeof(stringIn0));
	TEST_ASSERT_EQUAL_INT(0x00000000, dwordOut); // = Good
	TEST_ASSERT_EQUAL_STRING("Test 8= HistoryWrite", stringIn0);

	strcpy(stringIn0, "Test ");
	dwordOut = BrbUaAddEventNotifierText(9, stringIn0, sizeof(stringIn0));
	TEST_ASSERT_EQUAL_INT(0x00000000, dwordOut); // = Good
	TEST_ASSERT_EQUAL_STRING("Test 9= Subscribe, HistoryWrite", stringIn0);

	strcpy(stringIn0, "Test ");
	dwordOut = BrbUaAddEventNotifierText(10, stringIn0, sizeof(stringIn0));
	TEST_ASSERT_EQUAL_INT(0x00000000, dwordOut); // = Good
	TEST_ASSERT_EQUAL_STRING("Test 10= HistoryWrite", stringIn0);

	strcpy(stringIn0, "Test ");
	dwordOut = BrbUaAddEventNotifierText(11, stringIn0, sizeof(stringIn0));
	TEST_ASSERT_EQUAL_INT(0x00000000, dwordOut); // = Good
	TEST_ASSERT_EQUAL_STRING("Test 11= Subscribe, HistoryWrite", stringIn0);

	strcpy(stringIn0, "Test ");
	dwordOut = BrbUaAddEventNotifierText(12, stringIn0, sizeof(stringIn0));
	TEST_ASSERT_EQUAL_INT(0x00000000, dwordOut); // = Good
	TEST_ASSERT_EQUAL_STRING("Test 12= HistoryRead, HistoryWrite", stringIn0);

	strcpy(stringIn0, "Test ");
	dwordOut = BrbUaAddEventNotifierText(13, stringIn0, sizeof(stringIn0));
	TEST_ASSERT_EQUAL_INT(0x00000000, dwordOut); // = Good
	TEST_ASSERT_EQUAL_STRING("Test 13= Subscribe, HistoryRead, HistoryWrite", stringIn0);

	strcpy(stringIn0, "Test ");
	dwordOut = BrbUaAddEventNotifierText(14, stringIn0, sizeof(stringIn0));
	TEST_ASSERT_EQUAL_INT(0x00000000, dwordOut); // = Good
	TEST_ASSERT_EQUAL_STRING("Test 14= HistoryRead, HistoryWrite", stringIn0);

	strcpy(stringIn0, "Test ");
	dwordOut = BrbUaAddEventNotifierText(15, stringIn0, sizeof(stringIn0));
	TEST_ASSERT_EQUAL_INT(0x00000000, dwordOut); // = Good
	TEST_ASSERT_EQUAL_STRING("Test 15= Subscribe, HistoryRead, HistoryWrite", stringIn0);

	// Finished
	TEST_DONE;
}

// NOLINTEND(readability-*, bugprone-easily-swappable-parameters, bugprone-branch-clone, clang-diagnostic-invalid-utf8, clang-diagnostic-invalid-source-encoding, clang-diagnostic-pointer-arith, clang-diagnostic-strict-prototypes, clang-diagnostic-bad-function-cast, clang-analyzer-security.insecureAPI.*, hicpp-uppercase-literal-suffix, cppcoreguidelines-*, performance-*)

/*
B+R UnitTest: This is generated code.
Do not edit! Do not move!
Description: UnitTest Testprogramm infrastructure (TestSet).
LastUpdated: 2023-04-20 09:47:06Z
By B+R UnitTest Helper Version: 2.0.1.59
*/
UNITTEST_FIXTURES(fixtures)
{
	new_TestFixture("BrbUaAddEventNotifierText_NulPtr", BrbUaAddEventNotifierText_NulPtr),
	new_TestFixture("BrbUaAddEventNotifierText_Add", BrbUaAddEventNotifierText_Add),
};

UNITTEST_CALLER_COMPLETE_EXPLICIT(Set_BrbUaAddEventNotifierText, "Set_BrbUaAddEventNotifierText", 0, 0, fixtures, 0, 0, 0);
```

### Program Logical/UnitTests/UtBrbLibUa/UtBrbUaVariantValues (ANSIC) - UnitTests

#### variables.var - Name the suite and add PVs for the program
```iecst
(********************************************************************
 * COPYRIGHT --
 ********************************************************************
 * Program: utTemplate_automated
 * File: variables.var
 * Author: -
 * Created: -
 ********************************************************************
 * Local variables of program utTemplate_automated
 ********************************************************************)
(*Describe the test*)
VAR
	Testsuite : UtMgrTestSuite := (Name:='BrbUaVariantValues',Description:='(Optional field)Template for use with helper tool. Reference or add this program in the package "TS_UnitTest_UpdateTestPrograms"',Type:=utMgrTEST_TYPE_C,MetaInformation:='(Optional field):To be filled');
END_VAR
(*Input variables for testing*)
VAR
	variantIn0 : UAVariantData;
	stringIn0 : STRING[256] := '';
END_VAR
(*Functionblock instances for testing*)
(*Output variables for testing*)
VAR
	dwordOut : DWORD;
END_VAR
```
